DATA_BLOCK "_2010LV100P01_AD"   // DB14357
TITLE = Instance DB Adapter Block: _2010LV100P01
{ S7_Optimized_Access := 'FALSE' }
AUTHOR : METIS
NAME : APPT_DB
VERSION : 8.0
// stored: InstanceOfName IUSYS_PAC3220V1_POWERMON
"IUSYS_PAC3220V1_POWERMON"
BEGIN
   INREF := 6156;
   NET := 106;
   NODE := 22;
   RAW_InPut.SD00 := 16#0000_0001;
   RAW_InPut.SD04 := 401.1395;
   RAW_InPut.SD08 := 401.1483;
   RAW_InPut.SD12 := 400.6243;
   RAW_InPut.SD16 := 176.0122;
   RAW_InPut.SD20 := 183.3011;
   RAW_InPut.SD24 := 179.5082;
   RAW_InPut.SD28 := 49.93077;
   RAW_InPut.SD32 := 124737.3;
   RAW_InPut.SD36 := 97399.13;
   RAW_InPut.SD40 := 16734.09;
   RAW_InPut.SD44 := 0.7808338;
   RAW_InPut.SD48 := 3.005806E+08;
   RAW_InPut.SD52 := 3.817564E+08;
END_DATA_BLOCK

DATA_BLOCK "_2015PU027U01_AD"   // DB14415
{ S7_Optimized_Access := 'FALSE' }
VERSION : 0.1
// stored: InstanceOfName IUSYS_INVT_PN_MOTOR
"IUSYS_INVT_PN_MOTOR"
BEGIN
   INREF := 10040;
   OUTREF := 10040;
   FUNCTYPE := 41;
   OPTIONS := 1;
   NET := 106;
   NODE := 75;
   MCC := TRUE;
   RDY := TRUE;
   OVL := TRUE;
   LSTP := TRUE;
   REM := TRUE;
   SSW := TRUE;
   TFA := TRUE;
   DRDY := TRUE;
   STALL := TRUE;
   EARTH := TRUE;
   UBAL := TRUE;
   GFA := TRUE;
   GWA := TRUE;
   BUSF := TRUE;
   DOPR := TRUE;
   RAW_Input.SB00_0 := TRUE;
   RAW_Input.SB00_6 := TRUE;
   RAW_Input.SB01 := 16#03;
   RAW_Input.SB17_0 := TRUE;
   RAW_Input.SB17_1 := TRUE;
   RAW_Output.CB01 := 16#06;
   RAW_Output.CW08 := 16#0001;
   IHK.DelSTR_Timer_PV := 1;
   IHK.DelSTR_Timer_Mem := 1;
   IHK.DelSTP_Timer_PV := 3;
   IHK.RES_Timer_PV := 2;
   IHK.RES_Timer_Mem := 2;
   IHK.ChgOverTime_PV := 1;
   IHK.CoastTimer_PV := 1;
   IHK.DelSTP_Timer_DN := TRUE;
   IHK.ChgOverTime_DN := TRUE;
   IHK.CoastTimer_DN := TRUE;
   IHK.AUX_DelSTR_Time := 1;
   IHK.CoastSTP := TRUE;
   IHK.No_Acyc := TRUE;
   IHK.Pulse._01 := TRUE;
   IHK.Pulse._02 := TRUE;
   AC.Ons_Read_Req := TRUE;
   AC.Motor_Data_99._06 := 100.0;
   AC.Motor_Data_99._09 := 100;
   AC.Motor_Data_99._10 := 100.0;
   AC._99_Status := 16#0000_0000;
   AC_Read_99_Migra.STATUS := 16#0000_0000;
   OUT.MCC := TRUE;
   OUT.RDY := TRUE;
   OUT.OVL := TRUE;
   OUT.LSTP := TRUE;
   OUT.REM := TRUE;
   OUT.SSW := TRUE;
   OUT.TFA := TRUE;
   OUT.DRDY := TRUE;
   OUT.STALL := TRUE;
   OUT.EARTH := TRUE;
   OUT.UBAL := TRUE;
   OUT.GFA := TRUE;
   OUT.GWA := TRUE;
   OUT.BUSF := TRUE;
   OUT.DOPR := TRUE;
END_DATA_BLOCK

DATA_BLOCK "_2015PU028U01_AD"   // DB14416
{ S7_Optimized_Access := 'FALSE' }
VERSION : 0.1
// stored: InstanceOfName IUSYS_INVT_PN_MOTOR
"IUSYS_INVT_PN_MOTOR"
BEGIN
   INREF := 10072;
   OUTREF := 10072;
   FUNCTYPE := 41;
   OPTIONS := 1;
   NET := 106;
   NODE := 76;
   MCC := TRUE;
   RDY := TRUE;
   OVL := TRUE;
   REM := TRUE;
   SSW := TRUE;
   TFA := TRUE;
   DRDY := TRUE;
   STALL := TRUE;
   EARTH := TRUE;
   UBAL := TRUE;
   GFA := TRUE;
   GWA := TRUE;
   DTEST := TRUE;
   RAW_Output.CB01 := 16#06;
   RAW_Output.CW08 := 16#0001;
   IHK.DelSTR_Timer_PV := 1;
   IHK.DelSTR_Timer_Mem := 1;
   IHK.DelSTP_Timer_PV := 3;
   IHK.RES_Timer_PV := 2;
   IHK.RES_Timer_Mem := 2;
   IHK.ChgOverTime_PV := 1;
   IHK.CoastTimer_PV := 1;
   IHK.DelSTP_Timer_DN := TRUE;
   IHK.ChgOverTime_DN := TRUE;
   IHK.CoastTimer_DN := TRUE;
   IHK.AUX_DelSTR_Time := 1;
   IHK.CoastSTP := TRUE;
   IHK.No_Acyc := TRUE;
   IHK.Pulse._01 := TRUE;
   IHK.Pulse._02 := TRUE;
   AC.Ons_Read_Req := TRUE;
   AC.Motor_Data_99._06 := 100.0;
   AC.Motor_Data_99._09 := 100;
   AC.Motor_Data_99._10 := 100.0;
   AC._99_Status := 16#0000_0000;
   AC_Read_99_Migra.STATUS := 16#0000_0000;
   OUT.MCC := TRUE;
   OUT.RDY := TRUE;
   OUT.OVL := TRUE;
   OUT.REM := TRUE;
   OUT.SSW := TRUE;
   OUT.TFA := TRUE;
   OUT.DRDY := TRUE;
   OUT.STALL := TRUE;
   OUT.EARTH := TRUE;
   OUT.UBAL := TRUE;
   OUT.GFA := TRUE;
   OUT.GWA := TRUE;
   OUT.DTEST := TRUE;
END_DATA_BLOCK

DATA_BLOCK "_2015PU040U01_AD"   // DB14419
{ S7_Optimized_Access := 'FALSE' }
AUTHOR : FLSmidth
FAMILY : IUSYS
NAME : ADAPTOR
VERSION : 2.2
// stored: InstanceOfName IUSYS_ACS880_PN_MOTOR
"IUSYS_ACS880_PN_MOTOR"
BEGIN
   INREF := 10248;
   OUTREF := 10248;
   FUNCTYPE := 41;
   OPTIONS := 1;
   NET := 106;
   NODE := 16;
   CV := 100.0;
   MCC := TRUE;
   RDY := TRUE;
   OVL := TRUE;
   REM := TRUE;
   SSW := TRUE;
   TFA := TRUE;
   STALL := TRUE;
   EARTH := TRUE;
   UBAL := TRUE;
   GFA := TRUE;
   GWA := TRUE;
   BUSF := TRUE;
   DOPR := TRUE;
   RAW_Input.SB00_1 := TRUE;
   RAW_Input.SB00_4 := TRUE;
   RAW_Input.SB01_0 := TRUE;
   RAW_Input.SB01_4 := TRUE;
   RAW_Input.SB01_5 := TRUE;
   RAW_Input.SD04 := 16#0000_0000;
   RAW_Input.SD08 := 16#0000_0000;
   RAW_Input.SB16_7 := TRUE;
   RAW_Input.SW18 := 16#0B5E;
   RAW_Input.SW20 := 16#02AF;
   RAW_Output.CB00_2 := TRUE;
   RAW_Output.CB01_1 := TRUE;
   RAW_Output.CB01_2 := TRUE;
   RAW_Output.CB01_4 := TRUE;
   RAW_Output.CB01_5 := TRUE;
   RAW_Output.CB01_6 := TRUE;
   RAW_Output.CW02 := 16#4E20;
   RAW_Output.CW08 := 16#0001;
   IHK.DelSTR_Timer_PV := 1;
   IHK.DelSTR_Timer_Mem := 1;
   IHK.DelSTP_Timer_PV := 3;
   IHK.RES_Timer_PV := 2;
   IHK.RES_Timer_Mem := 2;
   IHK.ChgOverTime_PV := 1;
   IHK.CoastTimer_PV := 1;
   IHK.DelSTP_Timer_DN := TRUE;
   IHK.ChgOverTime_DN := TRUE;
   IHK.CoastTimer_DN := TRUE;
   IHK.AUX_DelSTR_Time := 1;
   IHK.CoastSTP := TRUE;
   IHK.No_Acyc := TRUE;
   IHK.Pulse._01 := TRUE;
   IHK.Pulse._02 := TRUE;
   AC.Ons_Read_Req := TRUE;
   AC._99_Status := 16#0000_0000;
   AC_Read_99_Migra.STATUS := 16#0000_0000;
   OUT.MCC := TRUE;
   OUT.RDY := TRUE;
   OUT.OVL := TRUE;
   OUT.REM := TRUE;
   OUT.SSW := TRUE;
   OUT.TFA := TRUE;
   OUT.STALL := TRUE;
   OUT.EARTH := TRUE;
   OUT.UBAL := TRUE;
   OUT.GFA := TRUE;
   OUT.GWA := TRUE;
   OUT.BUSF := TRUE;
   OUT.DOPR := TRUE;
END_DATA_BLOCK

DATA_BLOCK "_2015PU041U01_AD"   // DB14420
{ S7_Optimized_Access := 'FALSE' }
AUTHOR : FLSmidth
FAMILY : IUSYS
NAME : ADAPTOR
VERSION : 2.2
// stored: InstanceOfName IUSYS_ACS880_PN_MOTOR
"IUSYS_ACS880_PN_MOTOR"
BEGIN
   INREF := 10272;
   OUTREF := 10272;
   FUNCTYPE := 41;
   OPTIONS := 1;
   NET := 106;
   NODE := 78;
   CV := 100.0;
   MCC := TRUE;
   RDY := TRUE;
   OVL := TRUE;
   REM := TRUE;
   SSW := TRUE;
   TFA := TRUE;
   STALL := TRUE;
   EARTH := TRUE;
   UBAL := TRUE;
   GFA := TRUE;
   GWA := TRUE;
   BUSF := TRUE;
   DOPR := TRUE;
   RAW_Input.SB00_1 := TRUE;
   RAW_Input.SB00_4 := TRUE;
   RAW_Input.SB01_0 := TRUE;
   RAW_Input.SB01_4 := TRUE;
   RAW_Input.SB01_5 := TRUE;
   RAW_Input.SD04 := 16#0000_0000;
   RAW_Input.SD08 := 16#0000_0000;
   RAW_Input.SB16_7 := TRUE;
   RAW_Input.SW18 := 16#0B5E;
   RAW_Input.SW20 := 16#02AF;
   RAW_Output.CB00_2 := TRUE;
   RAW_Output.CB01_1 := TRUE;
   RAW_Output.CB01_2 := TRUE;
   RAW_Output.CB01_4 := TRUE;
   RAW_Output.CB01_5 := TRUE;
   RAW_Output.CB01_6 := TRUE;
   RAW_Output.CW02 := 16#4E20;
   RAW_Output.CW08 := 16#0001;
   IHK.DelSTR_Timer_PV := 1;
   IHK.DelSTR_Timer_Mem := 1;
   IHK.DelSTP_Timer_PV := 3;
   IHK.RES_Timer_PV := 2;
   IHK.RES_Timer_Mem := 2;
   IHK.ChgOverTime_PV := 1;
   IHK.CoastTimer_PV := 1;
   IHK.DelSTP_Timer_DN := TRUE;
   IHK.ChgOverTime_DN := TRUE;
   IHK.CoastTimer_DN := TRUE;
   IHK.AUX_DelSTR_Time := 1;
   IHK.CoastSTP := TRUE;
   IHK.No_Acyc := TRUE;
   IHK.Pulse._01 := TRUE;
   IHK.Pulse._02 := TRUE;
   AC.Ons_Read_Req := TRUE;
   AC._99_Status := 16#0000_0000;
   AC_Read_99_Migra.STATUS := 16#0000_0000;
   OUT.MCC := TRUE;
   OUT.RDY := TRUE;
   OUT.OVL := TRUE;
   OUT.REM := TRUE;
   OUT.SSW := TRUE;
   OUT.TFA := TRUE;
   OUT.STALL := TRUE;
   OUT.EARTH := TRUE;
   OUT.UBAL := TRUE;
   OUT.GFA := TRUE;
   OUT.GWA := TRUE;
   OUT.BUSF := TRUE;
   OUT.DOPR := TRUE;
END_DATA_BLOCK

DATA_BLOCK "_2015PU042U01_AD"   // DB14421
{ S7_Optimized_Access := 'FALSE' }
AUTHOR : FLSmidth
FAMILY : IUSYS
NAME : ADAPTOR
VERSION : 5.2
// stored: InstanceOfName IUSYS_3UF70_V5_MOTOR
"IUSYS_3UF70_V5_MOTOR"
BEGIN
   INREF := 7590;
   OUTREF := 7480;
   FUNCTYPE := 41;
   NET := 106;
   NODE := 64;
   MCC := TRUE;
   RDY := TRUE;
   OVL := TRUE;
   LSTP := TRUE;
   REM := TRUE;
   SSW := TRUE;
   TFA := TRUE;
   DRDY := TRUE;
   STALL := TRUE;
   EARTH := TRUE;
   UBAL := TRUE;
   GFA := TRUE;
   GWA := TRUE;
   BUSF := TRUE;
   DOPR := TRUE;
   ES := TRUE;
   Raw_InPut.SB00_1 := TRUE;
   Raw_InPut.SB00_2 := TRUE;
   Raw_InPut.SB00_3 := TRUE;
   Raw_InPut.SB01_3 := TRUE;
   Raw_OutPut.CB00_3 := TRUE;
   Raw_OutPut.CB00_7 := TRUE;
   OUT.MCC := TRUE;
   OUT.RDY := TRUE;
   OUT.OVL := TRUE;
   OUT.LSTP := TRUE;
   OUT.REM := TRUE;
   OUT.SSW := TRUE;
   OUT.TFA := TRUE;
   OUT.DRDY := TRUE;
   OUT.STALL := TRUE;
   OUT.EARTH := TRUE;
   OUT.UBAL := TRUE;
   OUT.GFA := TRUE;
   OUT.GWA := TRUE;
   OUT.BUSF := TRUE;
   OUT.DOPR := TRUE;
   OUT.ES := TRUE;
END_DATA_BLOCK

DATA_BLOCK "_MTR_SPARE_AD"   // DB14422
{ S7_Optimized_Access := 'FALSE' }
VERSION : 0.1
// stored: InstanceOfName IUSYS_ALTIVAR_PN_MOTOR
"IUSYS_ALTIVAR_PN_MOTOR"
BEGIN
END_DATA_BLOCK

DATA_BLOCK "_2015PU035U01_AD"   // DB14433
{ S7_Optimized_Access := 'FALSE' }
VERSION : 0.1
// stored: InstanceOfName IUSYS_INVT_PN_MOTOR
"IUSYS_INVT_PN_MOTOR"
BEGIN
   INREF := 10104;
   OUTREF := 10104;
   FUNCTYPE := 41;
   OPTIONS := 1;
   NET := 106;
   NODE := 75;
   CV := 20.0;
   MCC := TRUE;
   RDY := TRUE;
   OVL := TRUE;
   LSTP := TRUE;
   REM := TRUE;
   SSW := TRUE;
   TFA := TRUE;
   DRDY := TRUE;
   STALL := TRUE;
   EARTH := TRUE;
   UBAL := TRUE;
   GFA := TRUE;
   GWA := TRUE;
   BUSF := TRUE;
   DOPR := TRUE;
   RAW_Input.SB00_0 := TRUE;
   RAW_Input.SB00_6 := TRUE;
   RAW_Input.SB01 := 16#03;
   RAW_Input.SB17_0 := TRUE;
   RAW_Input.SB17_1 := TRUE;
   RAW_Output.CB01 := 16#06;
   RAW_Output.CW02 := 16#03E8;
   RAW_Output.CW08 := 16#0001;
   IHK.DelSTR_Timer_PV := 1;
   IHK.DelSTR_Timer_Mem := 1;
   IHK.DelSTP_Timer_PV := 3;
   IHK.RES_Timer_PV := 2;
   IHK.RES_Timer_Mem := 2;
   IHK.ChgOverTime_PV := 1;
   IHK.CoastTimer_PV := 1;
   IHK.DelSTP_Timer_DN := TRUE;
   IHK.ChgOverTime_DN := TRUE;
   IHK.CoastTimer_DN := TRUE;
   IHK.AUX_DelSTR_Time := 1;
   IHK.CoastSTP := TRUE;
   IHK.No_Acyc := TRUE;
   IHK.Pulse._01 := TRUE;
   IHK.Pulse._02 := TRUE;
   AC.Ons_Read_Req := TRUE;
   AC.Motor_Data_99._06 := 100.0;
   AC.Motor_Data_99._09 := 100;
   AC.Motor_Data_99._10 := 100.0;
   AC._99_Status := 16#0000_0000;
   AC_Read_99_Migra.STATUS := 16#0000_0000;
   OUT.MCC := TRUE;
   OUT.RDY := TRUE;
   OUT.OVL := TRUE;
   OUT.LSTP := TRUE;
   OUT.REM := TRUE;
   OUT.SSW := TRUE;
   OUT.TFA := TRUE;
   OUT.DRDY := TRUE;
   OUT.STALL := TRUE;
   OUT.EARTH := TRUE;
   OUT.UBAL := TRUE;
   OUT.GFA := TRUE;
   OUT.GWA := TRUE;
   OUT.BUSF := TRUE;
   OUT.DOPR := TRUE;
END_DATA_BLOCK

DATA_BLOCK "__2010CV300U01_AD"   // DB24007
{ S7_Optimized_Access := 'FALSE' }
VERSION : 0.1
// stored: InstanceOfName IUSYS_ACS880_PN_MOTOR
"IUSYS_ACS880_PN_MOTOR"
BEGIN
END_DATA_BLOCK

DATA_BLOCK "IUSYS_ALTIVAR_PN_MOTOR_DB_1"   // DB24011
{ S7_Optimized_Access := 'FALSE' }
VERSION : 0.1
// stored: InstanceOfName IUSYS_ALTIVAR_PN_MOTOR
"IUSYS_ALTIVAR_PN_MOTOR"
BEGIN
END_DATA_BLOCK

DATA_BLOCK "IUSYS_ALTIVAR_PN_MOTOR_DB"   // DB24012
{ S7_Optimized_Access := 'FALSE' }
VERSION : 0.1
// stored: InstanceOfName IUSYS_ALTIVAR_PN_MOTOR
"IUSYS_ALTIVAR_PN_MOTOR"
BEGIN
END_DATA_BLOCK

// folder: Modbus

DATA_BLOCK "MB_DATA_TEST"   // DB20
{ S7_Optimized_Access := 'FALSE' }
VERSION : 0.1
   VAR
      d12 : Word;
      d11 : Word;
      d10 : Word;
      d9 : Word;
      d8 : Word;
      d7 : Word;
      d6 : Word;
      d5 : Word;
      d4 : Word;
      d3 : Word;
      d2 : Word;
      d1 : Word;
   END_VAR
BEGIN
END_DATA_BLOCK

DATA_BLOCK "DB_DATA_MB_RD_VSD110"   // DB27
{ S7_Optimized_Access := 'FALSE' }
VERSION : 0.1
   VAR
      Frame1 : Struct
         REQ : Bool := TRUE;
         DISCONNECT : Bool := FALSE;
         CONNECT : TCON_IP_v4;
         DONE : Bool := TRUE;
         BUSY : Bool := FALSE;
         ERROR : Bool := FALSE;
         STATUS : Word := 16#0000;
         STATUS_SAVE : Word := 16#80C4;
         MB_MODE : USInt := 0;
         MB_DATA_ADDR : UDInt := 403202;
         MB_DATA_LEN : UInt := 8;
         MB_DATA_PTR : Array[0..10] of Int;
      END_STRUCT;
      Frame2 : Struct
         REQ : Bool := TRUE;
         DISCONNECT : Bool := FALSE;
         CONNECT : TCON_IP_v4;
         DONE : Bool := FALSE;
         BUSY : Bool := FALSE;
         ERROR : Bool := FALSE;
         STATUS : Word := 16#7004;
         STATUS_SAVE : Word := 16#8383;
         MB_MODE : USInt := 0;
         MB_DATA_ADDR : UDInt := 403105;
         MB_DATA_LEN : UInt := 2;
         MB_DATA_PTR : Array[0..10] of Int;
      END_STRUCT;
      Frame3 : Struct
         REQ : Bool := TRUE;
         DISCONNECT : Bool := FALSE;
         CONNECT : TCON_IP_v4;
         DONE : Bool := FALSE;
         BUSY : Bool := FALSE;
         ERROR : Bool := FALSE;
         STATUS : Word := 16#7004;
         STATUS_SAVE : Word := 16#80C6;
         MB_MODE : USInt := 0;
         MB_DATA_ADDR : UDInt := 407201;
         MB_DATA_LEN : UInt := 2;
         MB_DATA_PTR : Array[0..10] of Int;
      END_STRUCT;
      Frame4 : Struct
         REQ : Bool := TRUE;
         DISCONNECT : Bool := FALSE;
         CONNECT : TCON_IP_v4;
         DONE : Bool := FALSE;
         BUSY : Bool := FALSE;
         ERROR : Bool := FALSE;
         STATUS : Word := 16#7004;
         STATUS_SAVE : Word := 16#80C6;
         MB_MODE : USInt := 0;
         MB_DATA_ADDR : UDInt := 415323;
         MB_DATA_LEN : UInt := 2;
         MB_DATA_PTR : Array[0..10] of Int;
      END_STRUCT;
      Frame5 : Struct
         REQ : Bool := TRUE;
         DISCONNECT : Bool := FALSE;
         CONNECT : TCON_IP_v4;
         DONE : Bool := FALSE;
         BUSY : Bool := FALSE;
         ERROR : Bool := FALSE;
         STATUS : Word := 16#7000;
         STATUS_SAVE : Word := 16#8200;
         MB_MODE : USInt := 2;
         MB_DATA_ADDR : UDInt := 408502;
         MB_DATA_LEN : UInt := 2;
         MB_DATA_PTR : Array[0..10] of Int;
      END_STRUCT;
   END_VAR
BEGIN
   Frame1.CONNECT.LocalPort := 0;
   Frame1.CONNECT.RemotePort := 502;
   Frame1.CONNECT.RemoteAddress.ADDR[4] := 16#14;
   Frame1.CONNECT.RemoteAddress.ADDR[3] := 16#E7;
   Frame1.CONNECT.RemoteAddress.ADDR[2] := 16#1A;
   Frame1.CONNECT.RemoteAddress.ADDR[1] := 16#0A;
   Frame1.CONNECT.ActiveEstablished := TRUE;
   Frame1.CONNECT.ConnectionType := 16#0B;
   Frame1.CONNECT.ID := 16#0001;
   Frame1.CONNECT.InterfaceId := 64;
   Frame1.MB_DATA_PTR[0] := 3;
   Frame4.MB_DATA_PTR[10] := 0;
   Frame4.MB_DATA_PTR[9] := -32768;
   Frame4.MB_DATA_PTR[8] := 40;
   Frame4.MB_DATA_PTR[7] := 0;
   Frame4.MB_DATA_PTR[6] := 2391;
   Frame4.MB_DATA_PTR[5] := 6;
   Frame4.MB_DATA_PTR[4] := 0;
   Frame4.MB_DATA_PTR[3] := 0;
   Frame4.MB_DATA_PTR[2] := 0;
   Frame1.MB_DATA_PTR[8] := 40;
   Frame1.MB_DATA_PTR[7] := 0;
   Frame1.MB_DATA_PTR[6] := 4077;
   Frame1.MB_DATA_PTR[5] := 2;
   Frame1.MB_DATA_PTR[4] := 0;
   Frame1.MB_DATA_PTR[3] := 0;
   Frame1.MB_DATA_PTR[2] := 200;
   Frame1.MB_DATA_PTR[1] := 0;
   Frame1.MB_DATA_PTR[9] := -32768;
   Frame1.MB_DATA_PTR[10] := 0;
   Frame4.MB_DATA_PTR[1] := 0;
   Frame2.MB_DATA_PTR[10] := 0;
   Frame2.MB_DATA_PTR[9] := -32768;
   Frame2.MB_DATA_PTR[8] := 40;
   Frame2.MB_DATA_PTR[7] := 0;
   Frame2.MB_DATA_PTR[6] := 2391;
   Frame2.MB_DATA_PTR[5] := 0;
   Frame2.MB_DATA_PTR[4] := 0;
   Frame2.MB_DATA_PTR[3] := 0;
   Frame2.MB_DATA_PTR[2] := 0;
   Frame2.MB_DATA_PTR[1] := 200;
   Frame2.MB_DATA_PTR[0] := 500;
   Frame4.MB_DATA_PTR[0] := 1;
   Frame4.CONNECT.ID := 16#0004;
   Frame4.CONNECT.InterfaceId := 64;
   Frame3.MB_DATA_PTR[10] := 0;
   Frame3.MB_DATA_PTR[9] := -32768;
   Frame3.MB_DATA_PTR[8] := 40;
   Frame3.MB_DATA_PTR[7] := 0;
   Frame3.MB_DATA_PTR[6] := 2391;
   Frame3.MB_DATA_PTR[5] := 6;
   Frame3.MB_DATA_PTR[4] := 0;
   Frame3.MB_DATA_PTR[3] := 0;
   Frame3.MB_DATA_PTR[2] := 125;
   Frame3.MB_DATA_PTR[1] := 150;
   Frame3.MB_DATA_PTR[0] := 150;
   Frame4.CONNECT.LocalPort := 0;
   Frame4.CONNECT.RemotePort := 502;
   Frame4.CONNECT.RemoteAddress.ADDR[4] := 16#14;
   Frame4.CONNECT.RemoteAddress.ADDR[3] := 16#E7;
   Frame4.CONNECT.RemoteAddress.ADDR[2] := 16#1A;
   Frame4.CONNECT.RemoteAddress.ADDR[1] := 16#0A;
   Frame4.CONNECT.ActiveEstablished := TRUE;
   Frame4.CONNECT.ConnectionType := 16#0B;
   Frame2.CONNECT.LocalPort := 0;
   Frame2.CONNECT.RemotePort := 502;
   Frame2.CONNECT.RemoteAddress.ADDR[4] := 16#14;
   Frame2.CONNECT.RemoteAddress.ADDR[3] := 16#E7;
   Frame2.CONNECT.RemoteAddress.ADDR[2] := 16#1A;
   Frame2.CONNECT.RemoteAddress.ADDR[1] := 16#0A;
   Frame2.CONNECT.ActiveEstablished := TRUE;
   Frame2.CONNECT.ConnectionType := 16#0B;
   Frame2.CONNECT.ID := 16#0002;
   Frame2.CONNECT.InterfaceId := 64;
   Frame3.CONNECT.LocalPort := 0;
   Frame3.CONNECT.RemotePort := 502;
   Frame3.CONNECT.RemoteAddress.ADDR[4] := 16#14;
   Frame3.CONNECT.RemoteAddress.ADDR[3] := 16#E7;
   Frame3.CONNECT.RemoteAddress.ADDR[2] := 16#1A;
   Frame3.CONNECT.RemoteAddress.ADDR[1] := 16#0A;
   Frame3.CONNECT.ActiveEstablished := TRUE;
   Frame3.CONNECT.ConnectionType := 16#0B;
   Frame3.CONNECT.ID := 16#0003;
   Frame3.CONNECT.InterfaceId := 64;
   Frame5.CONNECT.InterfaceId := 64;
   Frame5.CONNECT.ID := 16#0005;
   Frame5.CONNECT.ConnectionType := 16#0B;
   Frame5.CONNECT.ActiveEstablished := TRUE;
   Frame5.CONNECT.RemoteAddress.ADDR[1] := 16#0A;
   Frame5.CONNECT.RemoteAddress.ADDR[2] := 16#1A;
   Frame5.CONNECT.RemoteAddress.ADDR[3] := 16#E7;
   Frame5.CONNECT.RemoteAddress.ADDR[4] := 16#14;
   Frame5.CONNECT.RemotePort := 502;
   Frame5.CONNECT.LocalPort := 0;
   Frame5.MB_DATA_PTR[0] := 0;
   Frame5.MB_DATA_PTR[1] := 125;
   Frame5.MB_DATA_PTR[2] := 125;
   Frame5.MB_DATA_PTR[3] := 0;
   Frame5.MB_DATA_PTR[4] := 0;
   Frame5.MB_DATA_PTR[5] := 6;
   Frame5.MB_DATA_PTR[6] := 2391;
   Frame5.MB_DATA_PTR[7] := 0;
   Frame5.MB_DATA_PTR[8] := 40;
   Frame5.MB_DATA_PTR[9] := -32768;
   Frame5.MB_DATA_PTR[10] := 0;
END_DATA_BLOCK

DATA_BLOCK "DB_DATA_MB_RD_VSD130_t"   // DB28
{ S7_Optimized_Access := 'FALSE' }
VERSION : 0.1
   VAR
      Frame1 : Struct
         REQ : Bool := TRUE;
         DISCONNECT : Bool := FALSE;
         CONNECT : TCON_IP_v4;
         DONE : Bool := FALSE;
         BUSY : Bool := FALSE;
         ERROR : Bool := FALSE;
         STATUS : Word := 16#7000;
         STATUS_SAVE : Word := 16#80C4;
         MB_MODE : USInt := 0;
         MB_DATA_ADDR : UDInt := 403202;
         MB_DATA_LEN : UInt := 8;
         MB_DATA_PTR : Array[0..10] of Int;
      END_STRUCT;
      Frame2 : Struct
         REQ : Bool := TRUE;
         DISCONNECT : Bool := FALSE;
         CONNECT : TCON_IP_v4;
         DONE : Bool := FALSE;
         BUSY : Bool := FALSE;
         ERROR : Bool := FALSE;
         STATUS : Word := 16#7000;
         STATUS_SAVE : Word := 16#80C6;
         MB_MODE : USInt := 0;
         MB_DATA_ADDR : UDInt := 403105;
         MB_DATA_LEN : UInt := 2;
         MB_DATA_PTR : Array[0..10] of Int;
      END_STRUCT;
      Frame3 : Struct
         REQ : Bool := FALSE;
         DISCONNECT : Bool := FALSE;
         CONNECT : TCON_IP_v4;
         DONE : Bool := FALSE;
         BUSY : Bool := FALSE;
         ERROR : Bool := FALSE;
         STATUS : Word := 16#7000;
         STATUS_SAVE : Word := 16#80C6;
         MB_MODE : USInt := 0;
         MB_DATA_ADDR : UDInt := 407201;
         MB_DATA_LEN : UInt := 2;
         MB_DATA_PTR : Array[0..10] of Int;
      END_STRUCT;
      Frame4 : Struct
         REQ : Bool := TRUE;
         DISCONNECT : Bool := FALSE;
         CONNECT : TCON_IP_v4;
         DONE : Bool := FALSE;
         BUSY : Bool := FALSE;
         ERROR : Bool := FALSE;
         STATUS : Word := 16#7000;
         STATUS_SAVE : Word := 16#80C6;
         MB_MODE : USInt := 0;
         MB_DATA_ADDR : UDInt := 415323;
         MB_DATA_LEN : UInt := 2;
         MB_DATA_PTR : Array[0..10] of Int;
      END_STRUCT;
      Frame5 : Struct
         REQ : Bool := TRUE;
         DISCONNECT : Bool := FALSE;
         CONNECT : TCON_IP_v4;
         DONE : Bool := FALSE;
         BUSY : Bool := FALSE;
         ERROR : Bool := FALSE;
         STATUS : Word := 16#7002;
         STATUS_SAVE : Word := 16#80C6;
         MB_MODE : USInt := 2;
         MB_DATA_ADDR : UDInt := 408502;
         MB_DATA_LEN : UInt := 2;
         MB_DATA_PTR : Array[0..10] of Int;
      END_STRUCT;
   END_VAR
BEGIN
   Frame1.CONNECT.LocalPort := 0;
   Frame1.CONNECT.RemotePort := 502;
   Frame1.CONNECT.RemoteAddress.ADDR[4] := 16#16;
   Frame1.CONNECT.RemoteAddress.ADDR[3] := 16#E7;
   Frame1.CONNECT.RemoteAddress.ADDR[2] := 16#1A;
   Frame1.CONNECT.RemoteAddress.ADDR[1] := 16#0A;
   Frame1.CONNECT.ActiveEstablished := TRUE;
   Frame1.CONNECT.ConnectionType := 16#0B;
   Frame1.CONNECT.ID := 16#0006;
   Frame1.CONNECT.InterfaceId := 64;
   Frame1.MB_DATA_PTR[0] := 545;
   Frame4.MB_DATA_PTR[10] := 0;
   Frame4.MB_DATA_PTR[9] := -32768;
   Frame4.MB_DATA_PTR[8] := 40;
   Frame4.MB_DATA_PTR[7] := 0;
   Frame4.MB_DATA_PTR[6] := 2391;
   Frame4.MB_DATA_PTR[5] := 6;
   Frame4.MB_DATA_PTR[4] := 0;
   Frame4.MB_DATA_PTR[3] := 0;
   Frame4.MB_DATA_PTR[2] := 0;
   Frame1.MB_DATA_PTR[8] := 0;
   Frame1.MB_DATA_PTR[7] := 0;
   Frame1.MB_DATA_PTR[6] := 0;
   Frame1.MB_DATA_PTR[5] := 2;
   Frame1.MB_DATA_PTR[4] := 0;
   Frame1.MB_DATA_PTR[3] := 0;
   Frame1.MB_DATA_PTR[2] := 500;
   Frame1.MB_DATA_PTR[1] := 0;
   Frame1.MB_DATA_PTR[9] := 0;
   Frame1.MB_DATA_PTR[10] := 0;
   Frame4.MB_DATA_PTR[1] := 3;
   Frame2.MB_DATA_PTR[10] := 0;
   Frame2.MB_DATA_PTR[9] := -32768;
   Frame2.MB_DATA_PTR[8] := 40;
   Frame2.MB_DATA_PTR[7] := 0;
   Frame2.MB_DATA_PTR[6] := 2391;
   Frame2.MB_DATA_PTR[5] := 0;
   Frame2.MB_DATA_PTR[4] := 0;
   Frame2.MB_DATA_PTR[3] := 0;
   Frame2.MB_DATA_PTR[2] := 0;
   Frame2.MB_DATA_PTR[1] := 0;
   Frame2.MB_DATA_PTR[0] := 500;
   Frame4.MB_DATA_PTR[0] := 0;
   Frame4.CONNECT.ID := 16#0009;
   Frame4.CONNECT.InterfaceId := 64;
   Frame3.MB_DATA_PTR[10] := 0;
   Frame3.MB_DATA_PTR[9] := -32768;
   Frame3.MB_DATA_PTR[8] := 40;
   Frame3.MB_DATA_PTR[7] := 0;
   Frame3.MB_DATA_PTR[6] := 0;
   Frame3.MB_DATA_PTR[5] := 6;
   Frame3.MB_DATA_PTR[4] := 0;
   Frame3.MB_DATA_PTR[3] := 0;
   Frame3.MB_DATA_PTR[2] := 0;
   Frame3.MB_DATA_PTR[1] := 150;
   Frame3.MB_DATA_PTR[0] := 0;
   Frame4.CONNECT.LocalPort := 0;
   Frame4.CONNECT.RemotePort := 502;
   Frame4.CONNECT.RemoteAddress.ADDR[4] := 16#16;
   Frame4.CONNECT.RemoteAddress.ADDR[3] := 16#E7;
   Frame4.CONNECT.RemoteAddress.ADDR[2] := 16#1A;
   Frame4.CONNECT.RemoteAddress.ADDR[1] := 16#0A;
   Frame4.CONNECT.ActiveEstablished := TRUE;
   Frame4.CONNECT.ConnectionType := 16#0B;
   Frame2.CONNECT.LocalPort := 0;
   Frame2.CONNECT.RemotePort := 502;
   Frame2.CONNECT.RemoteAddress.ADDR[4] := 16#16;
   Frame2.CONNECT.RemoteAddress.ADDR[3] := 16#E7;
   Frame2.CONNECT.RemoteAddress.ADDR[2] := 16#1A;
   Frame2.CONNECT.RemoteAddress.ADDR[1] := 16#0A;
   Frame2.CONNECT.ActiveEstablished := TRUE;
   Frame2.CONNECT.ConnectionType := 16#0B;
   Frame2.CONNECT.ID := 16#0007;
   Frame2.CONNECT.InterfaceId := 64;
   Frame3.CONNECT.LocalPort := 0;
   Frame3.CONNECT.RemotePort := 502;
   Frame3.CONNECT.RemoteAddress.ADDR[4] := 16#16;
   Frame3.CONNECT.RemoteAddress.ADDR[3] := 16#E7;
   Frame3.CONNECT.RemoteAddress.ADDR[2] := 16#1A;
   Frame3.CONNECT.RemoteAddress.ADDR[1] := 16#0A;
   Frame3.CONNECT.ActiveEstablished := TRUE;
   Frame3.CONNECT.ConnectionType := 16#0B;
   Frame3.CONNECT.ID := 16#0008;
   Frame3.CONNECT.InterfaceId := 64;
   Frame5.CONNECT.InterfaceId := 64;
   Frame5.CONNECT.ID := 16#000A;
   Frame5.CONNECT.ConnectionType := 16#0B;
   Frame5.CONNECT.ActiveEstablished := TRUE;
   Frame5.CONNECT.RemoteAddress.ADDR[1] := 16#0A;
   Frame5.CONNECT.RemoteAddress.ADDR[2] := 16#1A;
   Frame5.CONNECT.RemoteAddress.ADDR[3] := 16#E7;
   Frame5.CONNECT.RemoteAddress.ADDR[4] := 16#16;
   Frame5.CONNECT.RemotePort := 502;
   Frame5.CONNECT.LocalPort := 0;
   Frame5.MB_DATA_PTR[0] := 0;
   Frame5.MB_DATA_PTR[1] := 500;
   Frame5.MB_DATA_PTR[2] := 0;
   Frame5.MB_DATA_PTR[3] := 0;
   Frame5.MB_DATA_PTR[4] := 0;
   Frame5.MB_DATA_PTR[5] := 6;
   Frame5.MB_DATA_PTR[6] := 2391;
   Frame5.MB_DATA_PTR[7] := 0;
   Frame5.MB_DATA_PTR[8] := 40;
   Frame5.MB_DATA_PTR[9] := -32768;
   Frame5.MB_DATA_PTR[10] := 0;
END_DATA_BLOCK

DATA_BLOCK "VSD110"   // DB29
{ S7_Optimized_Access := 'TRUE' }
VERSION : 0.1
// stored: InstanceOfName Mgt_VSD_Com
"Mgt_VSD_Com"
BEGIN
   "Counter".CU := TRUE;
   "Counter".R := TRUE;
   "Counter".QD := TRUE;
   "Counter".PV := 1;
   Time_Value2 := 50;
   Time_Value3 := 50;
   Time_Value4 := 50;
   Time_Value5 := 50;
   Time_Value6 := 50;
   Time_Value7 := 50;
   Time_Value8 := 50;
   Time_Value9 := 50;
END_DATA_BLOCK

DATA_BLOCK "VSD130_t"   // DB30
{ S7_Optimized_Access := 'TRUE' }
VERSION : 0.1
// stored: InstanceOfName Mgt_VSD_Com
"Mgt_VSD_Com"
BEGIN
   "Counter".CU := TRUE;
   "Counter".R := TRUE;
   "Counter".QD := TRUE;
   "Counter".PV := 1;
   Time_Value2 := 50;
   Time_Value3 := 50;
   Time_Value4 := 50;
   Time_Value5 := 50;
   Time_Value6 := 50;
   Time_Value7 := 50;
   Time_Value8 := 50;
   Time_Value9 := 50;
   RD_3201_3208.MB_DATA_ADDR := 400001;
   RD_3201_3208.MB_DATA_LEN := 4;
   RD_3201_3208.STATUS := 16#7004;
   RD_3104_3105.MB_DATA_ADDR := 400004;
   RD_3104_3105.MB_DATA_LEN := 2;
   RD_3104_3105.STATUS := 16#7004;
   RD_7200_7201.MB_DATA_ADDR := 400005;
   RD_7200_7201.MB_DATA_LEN := 2;
   RD_7200_7201.STATUS := 16#7004;
   RD_15323.REQ := TRUE;
   RD_15323.MB_DATA_ADDR := 400007;
   RD_15323.MB_DATA_LEN := 2;
   RD_15323.BUSY := TRUE;
   RD_15323.STATUS := 16#7006;
   WR_8501_8502.DISCONNECT := TRUE;
   WR_8501_8502.MB_MODE := 2;
   WR_8501_8502.MB_DATA_ADDR := 40008;
   WR_8501_8502.MB_DATA_LEN := 2;
   WR_8501_8502.STATUS := 16#7000;
END_DATA_BLOCK

DATA_BLOCK "DB_DATA_MB_RD_VSD130"   // DB31
{ S7_Optimized_Access := 'FALSE' }
VERSION : 0.1
   VAR
      Frame1 : Struct
         REQ : Bool := TRUE;
         DISCONNECT : Bool := FALSE;
         CONNECT : TCON_IP_v4;
         DONE : Bool := FALSE;
         BUSY : Bool := FALSE;
         ERROR : Bool := FALSE;
         STATUS : Word := 16#7004;
         STATUS_SAVE : Word := 16#8383;
         MB_MODE : USInt := 0;
         MB_DATA_ADDR : UDInt := 403202;
         MB_DATA_LEN : UInt := 8;
         MB_DATA_PTR : Array[0..10] of Int;
      END_STRUCT;
      Frame2 : Struct
         REQ : Bool := TRUE;
         DISCONNECT : Bool := FALSE;
         CONNECT : TCON_IP_v4;
         DONE : Bool := FALSE;
         BUSY : Bool := FALSE;
         ERROR : Bool := FALSE;
         STATUS : Word := 16#7004;
         STATUS_SAVE : Word := 16#8383;
         MB_MODE : USInt := 0;
         MB_DATA_ADDR : UDInt := 403105;
         MB_DATA_LEN : UInt := 2;
         MB_DATA_PTR : Array[0..10] of Int;
      END_STRUCT;
      Frame3 : Struct
         REQ : Bool := TRUE;
         DISCONNECT : Bool := FALSE;
         CONNECT : TCON_IP_v4;
         DONE : Bool := TRUE;
         BUSY : Bool := FALSE;
         ERROR : Bool := FALSE;
         STATUS : Word := 16#0000;
         STATUS_SAVE : Word := 16#8383;
         MB_MODE : USInt := 0;
         MB_DATA_ADDR : UDInt := 407201;
         MB_DATA_LEN : UInt := 2;
         MB_DATA_PTR : Array[0..10] of Int;
      END_STRUCT;
      Frame4 : Struct
         REQ : Bool := TRUE;
         DISCONNECT : Bool := FALSE;
         CONNECT : TCON_IP_v4;
         DONE : Bool := FALSE;
         BUSY : Bool := FALSE;
         ERROR : Bool := FALSE;
         STATUS : Word := 16#7004;
         STATUS_SAVE : Word := 16#8383;
         MB_MODE : USInt := 0;
         MB_DATA_ADDR : UDInt := 415323;
         MB_DATA_LEN : UInt := 2;
         MB_DATA_PTR : Array[0..10] of Int;
      END_STRUCT;
      Frame5 : Struct
         REQ : Bool := TRUE;
         DISCONNECT : Bool := FALSE;
         CONNECT : TCON_IP_v4;
         DONE : Bool := FALSE;
         BUSY : Bool := FALSE;
         ERROR : Bool := FALSE;
         STATUS : Word := 16#7000;
         STATUS_SAVE : Word := 16#80C4;
         MB_MODE : USInt := 2;
         MB_DATA_ADDR : UDInt := 408502;
         MB_DATA_LEN : UInt := 2;
         MB_DATA_PTR : Array[0..10] of Int;
      END_STRUCT;
   END_VAR
BEGIN
   Frame1.CONNECT.LocalPort := 0;
   Frame1.CONNECT.RemotePort := 502;
   Frame1.CONNECT.RemoteAddress.ADDR[4] := 16#16;
   Frame1.CONNECT.RemoteAddress.ADDR[3] := 16#E7;
   Frame1.CONNECT.RemoteAddress.ADDR[2] := 16#1A;
   Frame1.CONNECT.RemoteAddress.ADDR[1] := 16#0A;
   Frame1.CONNECT.ActiveEstablished := TRUE;
   Frame1.CONNECT.ConnectionType := 16#0B;
   Frame1.CONNECT.ID := 16#0006;
   Frame1.CONNECT.InterfaceId := 64;
   Frame1.MB_DATA_PTR[0] := 545;
   Frame4.MB_DATA_PTR[10] := 0;
   Frame4.MB_DATA_PTR[9] := -32768;
   Frame4.MB_DATA_PTR[8] := 40;
   Frame4.MB_DATA_PTR[7] := 0;
   Frame4.MB_DATA_PTR[6] := 2391;
   Frame4.MB_DATA_PTR[5] := 6;
   Frame4.MB_DATA_PTR[4] := 0;
   Frame4.MB_DATA_PTR[3] := 0;
   Frame4.MB_DATA_PTR[2] := 0;
   Frame1.MB_DATA_PTR[8] := 40;
   Frame1.MB_DATA_PTR[7] := 0;
   Frame1.MB_DATA_PTR[6] := 0;
   Frame1.MB_DATA_PTR[5] := 2;
   Frame1.MB_DATA_PTR[4] := 0;
   Frame1.MB_DATA_PTR[3] := 0;
   Frame1.MB_DATA_PTR[2] := 500;
   Frame1.MB_DATA_PTR[1] := 0;
   Frame1.MB_DATA_PTR[9] := -32768;
   Frame1.MB_DATA_PTR[10] := 0;
   Frame4.MB_DATA_PTR[1] := 3;
   Frame2.MB_DATA_PTR[10] := 0;
   Frame2.MB_DATA_PTR[9] := -32768;
   Frame2.MB_DATA_PTR[8] := 40;
   Frame2.MB_DATA_PTR[7] := 0;
   Frame2.MB_DATA_PTR[6] := 2391;
   Frame2.MB_DATA_PTR[5] := 0;
   Frame2.MB_DATA_PTR[4] := 0;
   Frame2.MB_DATA_PTR[3] := 0;
   Frame2.MB_DATA_PTR[2] := 0;
   Frame2.MB_DATA_PTR[1] := 0;
   Frame2.MB_DATA_PTR[0] := 500;
   Frame4.MB_DATA_PTR[0] := 0;
   Frame4.CONNECT.ID := 16#0009;
   Frame4.CONNECT.InterfaceId := 64;
   Frame3.MB_DATA_PTR[10] := 0;
   Frame3.MB_DATA_PTR[9] := -32768;
   Frame3.MB_DATA_PTR[8] := 40;
   Frame3.MB_DATA_PTR[7] := 0;
   Frame3.MB_DATA_PTR[6] := 2391;
   Frame3.MB_DATA_PTR[5] := 6;
   Frame3.MB_DATA_PTR[4] := 0;
   Frame3.MB_DATA_PTR[3] := 0;
   Frame3.MB_DATA_PTR[2] := 125;
   Frame3.MB_DATA_PTR[1] := 150;
   Frame3.MB_DATA_PTR[0] := 0;
   Frame4.CONNECT.LocalPort := 0;
   Frame4.CONNECT.RemotePort := 502;
   Frame4.CONNECT.RemoteAddress.ADDR[4] := 16#16;
   Frame4.CONNECT.RemoteAddress.ADDR[3] := 16#E7;
   Frame4.CONNECT.RemoteAddress.ADDR[2] := 16#1A;
   Frame4.CONNECT.RemoteAddress.ADDR[1] := 16#0A;
   Frame4.CONNECT.ActiveEstablished := TRUE;
   Frame4.CONNECT.ConnectionType := 16#0B;
   Frame2.CONNECT.LocalPort := 0;
   Frame2.CONNECT.RemotePort := 502;
   Frame2.CONNECT.RemoteAddress.ADDR[4] := 16#16;
   Frame2.CONNECT.RemoteAddress.ADDR[3] := 16#E7;
   Frame2.CONNECT.RemoteAddress.ADDR[2] := 16#1A;
   Frame2.CONNECT.RemoteAddress.ADDR[1] := 16#0A;
   Frame2.CONNECT.ActiveEstablished := TRUE;
   Frame2.CONNECT.ConnectionType := 16#0B;
   Frame2.CONNECT.ID := 16#0007;
   Frame2.CONNECT.InterfaceId := 64;
   Frame3.CONNECT.LocalPort := 0;
   Frame3.CONNECT.RemotePort := 502;
   Frame3.CONNECT.RemoteAddress.ADDR[4] := 16#16;
   Frame3.CONNECT.RemoteAddress.ADDR[3] := 16#E7;
   Frame3.CONNECT.RemoteAddress.ADDR[2] := 16#1A;
   Frame3.CONNECT.RemoteAddress.ADDR[1] := 16#0A;
   Frame3.CONNECT.ActiveEstablished := TRUE;
   Frame3.CONNECT.ConnectionType := 16#0B;
   Frame3.CONNECT.ID := 16#0008;
   Frame3.CONNECT.InterfaceId := 64;
   Frame5.CONNECT.InterfaceId := 64;
   Frame5.CONNECT.ID := 16#000A;
   Frame5.CONNECT.ConnectionType := 16#0B;
   Frame5.CONNECT.ActiveEstablished := TRUE;
   Frame5.CONNECT.RemoteAddress.ADDR[1] := 16#0A;
   Frame5.CONNECT.RemoteAddress.ADDR[2] := 16#1A;
   Frame5.CONNECT.RemoteAddress.ADDR[3] := 16#E7;
   Frame5.CONNECT.RemoteAddress.ADDR[4] := 16#16;
   Frame5.CONNECT.RemotePort := 502;
   Frame5.CONNECT.LocalPort := 0;
   Frame5.MB_DATA_PTR[0] := 0;
   Frame5.MB_DATA_PTR[1] := 500;
   Frame5.MB_DATA_PTR[2] := 125;
   Frame5.MB_DATA_PTR[3] := 0;
   Frame5.MB_DATA_PTR[4] := 0;
   Frame5.MB_DATA_PTR[5] := 6;
   Frame5.MB_DATA_PTR[6] := 2391;
   Frame5.MB_DATA_PTR[7] := 0;
   Frame5.MB_DATA_PTR[8] := 40;
   Frame5.MB_DATA_PTR[9] := -32768;
   Frame5.MB_DATA_PTR[10] := 0;
END_DATA_BLOCK

DATA_BLOCK "VSD130_DB"   // DB32
{ S7_Optimized_Access := 'TRUE' }
VERSION : 0.1
// stored: InstanceOfName Mgt_VSD_Com
"Mgt_VSD_Com"
BEGIN
END_DATA_BLOCK

// folder: System blocks/Program resources

DATA_BLOCK "Speed_BC180_1"   // DB19
{ S7_Optimized_Access := 'TRUE' }
AUTHOR : Simatic
FAMILY : IEC
NAME : IEC_TMR
VERSION : 1.0
// stored: InstanceOfName IEC_TIMER
"IEC_TIMER"
BEGIN
END_DATA_BLOCK

DATA_BLOCK "Speed_BC180_2"   // DB21
{ S7_Optimized_Access := 'TRUE' }
AUTHOR : Simatic
FAMILY : IEC
NAME : IEC_TMR
VERSION : 1.0
// stored: InstanceOfName IEC_TIMER
"IEC_TIMER"
BEGIN
END_DATA_BLOCK

DATA_BLOCK "Speed_BC120_1"   // DB22
{ S7_Optimized_Access := 'TRUE' }
AUTHOR : Simatic
FAMILY : IEC
NAME : IEC_TMR
VERSION : 1.0
// stored: InstanceOfName IEC_TIMER
"IEC_TIMER"
BEGIN
END_DATA_BLOCK

DATA_BLOCK "Speed_BC120_2"   // DB23
{ S7_Optimized_Access := 'TRUE' }
AUTHOR : Simatic
FAMILY : IEC
NAME : IEC_TMR
VERSION : 1.0
// stored: InstanceOfName IEC_TIMER
"IEC_TIMER"
BEGIN
END_DATA_BLOCK

DATA_BLOCK "_2010SJ950M01_T1"   // DB24
{ S7_Optimized_Access := 'TRUE' }
AUTHOR : Simatic
FAMILY : IEC
NAME : IEC_TMR
VERSION : 1.0
// stored: InstanceOfName IEC_TIMER
"IEC_TIMER"
BEGIN
END_DATA_BLOCK

DATA_BLOCK "IEC_Timer_0_DB"   // DB50
{ S7_Optimized_Access := 'TRUE' }
AUTHOR : Simatic
FAMILY : IEC
NAME : IEC_TMR
VERSION : 1.0
// stored: InstanceOfName IEC_TIMER
"IEC_TIMER"
BEGIN
   ST := T#20D_8H_56M_38S_289MS;
   PT := T#2S;
END_DATA_BLOCK

// folder: (top level)

FUNCTION_BLOCK "LMNGEN_C"   // FB33, LAD
TITLE = PID : Output continuous PID controller
{ S7_Optimized_Access := 'FALSE' }
AUTHOR : MODIFIED
FAMILY : MODCONT
NAME : LMNGEN_C
VERSION : 1.0
   VAR_INPUT
      MAN : Real;   // manual value
      LMN_HLM : Real := 100.0;   // manipulated value high limit
      LMN_LLM : Real;   // manipulated value low limit
      LMN_URLM : Real := 10.0;   // manipulated value up rate limit
      LMN_DRLM : Real := 10.0;   // manipulated down rate limit
      DF_OUTV : Real;   // default output variable
      MAN_ON : Bool := TRUE;   // manual value on
      MANGN_ON : Bool;   // manual value generating on
      MANUP : Bool;   // manual value up
      MANDN : Bool;   // manual value down
      LMNRC_ON : Bool;   // manipulated value rate of change on
      DFOUT_ON : Bool;   // default output variable on
      COM_RST : Bool;   // complete restart
      CYCLE : Time := T#1S;   // sample time
      PID_LMNG : Struct
         PID_OUTV : Real;   // PID output variable
         PID_SCTR : Real;   // PID output variable for step controller
      END_STRUCT;
   END_VAR
   VAR_OUTPUT
      LMN : Real;   // manipulated value
      QLMN_HLM : Bool;   // high limit of manipulated value reached
      QLMN_LLM : Bool;   // low limit of manipulated value reached
      LMNG_PID : Struct
         LMN : Real;   // manipulated value
         LMN_HLM : Real;   // manipulated value high limit
         LMN_LLM : Real;   // manipulated value low limit
         R_MTR_TM : Real;   // motor manipulated value
         ARWHL_ON : Bool;   // anti reset wind-up in high limit on
         ARWLL_ON : Bool;   // anti reset wind-up in low limit on
         MAN_ON : Bool;   // manual mode on
         LMNGS_ON : Bool;   // PID-algorithm for step controller on
         LMNR_ON : Bool;   // repeated manipulated value on
      END_STRUCT;
   END_VAR
   VAR
      MP1 : Real;   // MP1: manipulated value
      LMN_OP : Real;   // manipulated value operation
      LMNOP_ON : Bool;   // manipulated value operation on
      stUpMan : Time;
      stDownMan : Time;
   END_VAR
   VAR_TEMP
      Hvar : Real;   // Hilfsvariable
      rCycle : Real;   // Abtastzeit in real
      Diff : Real;   // Änderungswert bei der Handwertbedienung
      RocHlm : Real;   // Obere Begrenzung im Hochlaufgeber
      RocLlm : Real;   // Untere Begrenzung im Hochlaufgeber
      Pid_Outv : Real;   // PID output variable
      dLmn : Real;   // Stellwert
      bLmnopOn : Bool;   // manipulated value operation on
      bCasOn : Bool;   // cascade mode on
      bArwhlOn : Bool;   // Anti Reset Wind-up high limit Bit für Struktur PID_LMNG
      bArwllOn : Bool;   // Anti Reset Wind-up low limit Bit für Struktur PID_LMNG
   END_VAR
BEGIN
END_FUNCTION_BLOCK

FUNCTION_BLOCK "PID"   // FB39, LAD
TITLE = PID: Output PID-algorithm
{ S7_Optimized_Access := 'FALSE' }
AUTHOR : MODIFIED
FAMILY : MODCONT
NAME : PID
VERSION : 1.1
   VAR_INPUT
      ER : Real;   // error-signal
      PV : Real;   // process variable
      GAIN : Real := 1.0;   // proportional gain
      TI : Time := T#20S;   // reset time
      I_ITLVAL : Real;   // initialization value of the integral action
      TD : Time := T#10S;   // derivative time
      TM_LAG : Time := T#2S;   // time lag of the derivative action
      DISV : Real;   // disturbance variable
      P_SEL : Bool := TRUE;   // proportional action selected
      PFDB_SEL : Bool;   // proportional action in feedback path selected
      DFDB_SEL : Bool;   // derivative action in feedback path on
      I_SEL : Bool := TRUE;   // integral action selected
      INT_HOLD : Bool;   // integral action hold
      I_ITL_ON : Bool;   // initialization of the integral action on
      D_SEL : Bool;   // derivative action selected
      DISV_SEL : Bool := TRUE;   // disturbance variable on
      COM_RST : Bool;   // complete restart
      CYCLE : Time := T#1S;   // sample time
      LMNG_PID : Struct
         LMN : Real;   // manipulated value
         LMN_HLM : Real;   // manipulated value high limit
         LMN_LLM : Real;   // manipulated value low limit
         R_MTR_TM : Real;   // motor manipulated value
         ARWHL_ON : Bool;   // anti reset wind-up in high limit on
         ARWLL_ON : Bool;   // anti reset wind-up in low limit on
         MAN_ON : Bool;   // manual mode on
         LMNGS_ON : Bool;   // PID-algorithm for step controller on
         LMNR_ON : Bool;   // repeated manipulated value on
      END_STRUCT;
   END_VAR
   VAR_OUTPUT
      LMN_P : Real;   // proportionality component
      LMN_I : Real;   // integral component
      LMN_D : Real;   // derivative component
      PID_LMNG : Struct
         PID_OUTV : Real;   // PID output variable
         PID_SCTR : Real;   // PID output variable for step controller
      END_STRUCT;
   END_VAR
   VAR
      sInvAlt : Real;
      sIanteilAlt : Real;
      sRestInt : Real;
      sRestDif : Real;
      sRueck : Real;
      sbILimOn : Bool := TRUE;
   END_VAR
   VAR_TEMP
      Hvar : Real;   // Hilfsvariable
      ErKp : Real;   // Variable ER*GAIN
      rTi : Real;   // Integrationszeit in real
      rTd : Real;   // Differentiationszeit in real
      rTmLag : Real;   // Verzögerungszeit in real
      rCycle : Real;   // Abtastzeit in real
      Panteil : Real;   // P-Anteil
      Ianteil : Real;   // I-Anteil
      Diff : Real;   // Änderungswert
      Danteil : Real;   // D-Anteil
      Verstaerk : Real;   // Verstärkung
      RueckDiff : Real;   // Differenz des Rückkopplungswertes
      RueckAlt : Real;   // Alter Rückkopplungswert
      dDisv : Real;   // disturbance variable
      dLmn : Real;   // Stellwert
      PidOutv : Real;   // PID-Ausgangswert
      PidSctr : Real;   // PID-Ausgangswert für Schrittregler
      rLmnHlm : Real;   // Obere Begrenzung
      rLmnLlm : Real;   // Untere Begrenzung
      rMtrTm : Real;   // Motorstellzeit
      bArwhlOn : Bool;   // anti reset wind-up in high limit on
      bArwllOn : Bool;   // anti reset wind-up in low limit on
      bManOn : Bool;   // manual mode on
      bLmngsOn : Bool;   // PID-algorithm for step controller
      bLmnrOn : Bool;   // step controller with repeated manipulated value
   END_VAR
BEGIN
END_FUNCTION_BLOCK

FUNCTION_BLOCK "Eqip_Maintenance"   // FB106, FBD
TITLE = Equipment Maintenance Hour Meter (5 sec)
{ S7_Optimized_Access := 'FALSE' }
VERSION : 0.1
   VAR_INPUT
      IN : Bool;   // Equipment (Motor) Status
      Reset_1 : Bool;   // Maintenance Done
      Reset_2 : Bool;   // Maintenance Done
      Reset_3 : Bool;   // Maintenance Done
      Reset_4 : Bool;   // Maintenance Done
   END_VAR
   VAR_OUTPUT
      Cnt_Hours_1 : DInt;   // Counter-1 of Hours
      Cnt_Hours_2 : DInt;   // Counter-2 of Hours
      Cnt_Hours_3 : DInt;   // Counter-3 of Hours
      Cnt_Hours_4 : DInt;   // Counter-4 of Hours
   END_VAR
   VAR
      Accum_1 : DInt;   // Accum_1 (sec)
      Accum_2 : DInt;   // Accum_2 (sec)
      Accum_3 : DInt;   // Accum_3 (sec)
      Accum_4 : DInt;   // Accum_4 (sec)
   END_VAR
   VAR_TEMP
      tmp_bool : Bool;
   END_VAR
BEGIN

REGION Network 1: Reset Seconds ACCUM_1
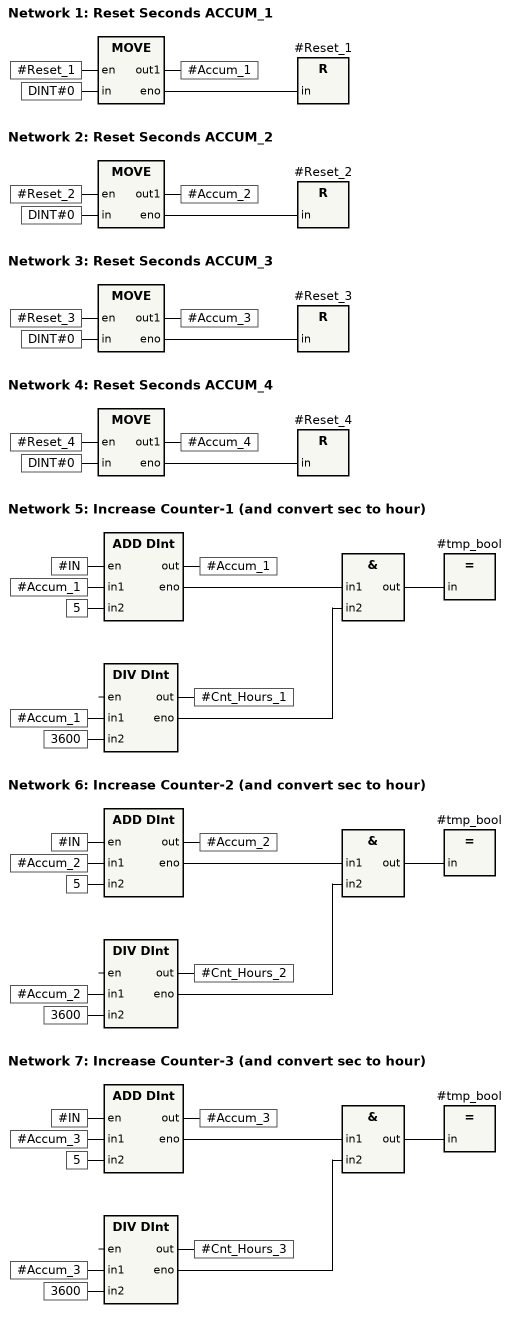
   IF #Reset_1 THEN
       #Accum_1 := DINT#0;
       #Reset_1 := FALSE;
   END_IF;
END_REGION

REGION Network 2: Reset Seconds ACCUM_2
   IF #Reset_2 THEN
       #Accum_2 := DINT#0;
       #Reset_2 := FALSE;
   END_IF;
END_REGION

REGION Network 3: Reset Seconds ACCUM_3
   IF #Reset_3 THEN
       #Accum_3 := DINT#0;
       #Reset_3 := FALSE;
   END_IF;
END_REGION

REGION Network 4: Reset Seconds ACCUM_4
   IF #Reset_4 THEN
       #Accum_4 := DINT#0;
       #Reset_4 := FALSE;
   END_IF;
END_REGION

REGION Network 5: Increase Counter-1 (and convert sec to hour)
   IF #IN THEN #Accum_1 := #Accum_1 + 5; END_IF;
   #Cnt_Hours_1 := #Accum_1 / 3600;
   #tmp_bool := #IN;
END_REGION

REGION Network 6: Increase Counter-2 (and convert sec to hour)
   IF #IN THEN #Accum_2 := #Accum_2 + 5; END_IF;
   #Cnt_Hours_2 := #Accum_2 / 3600;
   #tmp_bool := #IN;
END_REGION

REGION Network 7: Increase Counter-3 (and convert sec to hour)
   IF #IN THEN #Accum_3 := #Accum_3 + 5; END_IF;
   #Cnt_Hours_3 := #Accum_3 / 3600;
   #tmp_bool := #IN;
END_REGION

REGION Network 8: Increase Counter-4 (and convert sec to hour)
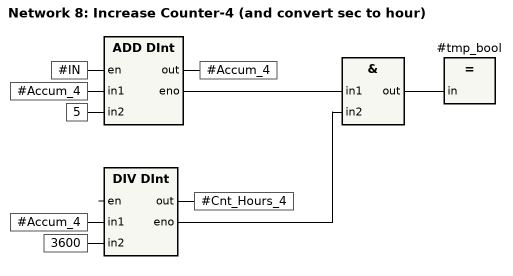
   IF #IN THEN #Accum_4 := #Accum_4 + 5; END_IF;
   #Cnt_Hours_4 := #Accum_4 / 3600;
   #tmp_bool := #IN;
END_REGION
END_FUNCTION_BLOCK

FUNCTION_BLOCK "ACESYS_MASTER"   // FB200, FBD
TITLE = ACESYS V8.0 - Build 001 - MASTER Block
{ S7_Optimized_Access := 'FALSE' }
AUTHOR : FLSmidth
FAMILY : ACESYS
NAME : MASTER
VERSION : 8.0
   VAR_INPUT
      LOC_TYPE : Bool;   // Accept return in local without command: "0"= Disable / "1" = Enable
      REM_TYPE : Bool;   // REM Switch Type : "0"= Normal / "1" = Force Local
      SIM_ENABLE : Bool;   // Enable Device Simulation : "0"= Disable / "1" = Enable
      SS_FP_ENABLE : Bool := TRUE;   // Enable Single Start from FP : "0"= Disable / "1" = Enable
      SS_Field_ENABLE : Bool := TRUE;   // Enable Single Start from Field: "0"= Disable / "1" = Enable
      MAN_ENABLE : Bool := TRUE;   // Enable Manual Mode : "0"= Disable / "1" = Enable
      LOC_ENABLE : Bool := TRUE;   // Enable Manual Local : "0"= Disable / "1" = Enable
      TEST_ENABLE : Bool := TRUE;   // Enable Test Mode : "0"= Disable / "1" = Enable
      QSTOP_FP_Unit : Bool;   // Enable Quick Stop from Unit FP: "0"= Disable / "1" = Enable
      RED_ENABLE : Bool;   // Redundant system : "0"= Disable / "1" = Enable
      WatchDog_HMI_Enable : Bool;   // Enable Watchdog Supervision : "0"= Disable / "1" = Enable
      WatchDog_HMI_Time : Time := T#30MS;   // WatchDog Time HMI
      OB1_CycleTime : Int;
   END_VAR
   VAR_OUTPUT
      WatchDog_HMI_Elap : Time;   // WatchDog HMI Elapsed Time
      MASTER_Link : "ACESYS_MASTER_LINK";   // Link to Departments
      First_Scan : Bool;   // First Scan Pulse
      SEC_Toggle : Bool;   // 1 Sec. Toggle
   END_VAR
   VAR_IN_OUT
      WatchDog_HMI : Bool;   // WatchDog Pulse from HMI
   END_VAR
   VAR
      BlockInfo : Struct
         Ace_Version : Int;   // Acesys Block Version Number
         Ace_BuildNo : Int;   // Acesys Block Build Number
         State_Act : Int;   // Actual State Number
         State_Prev : Int;   // Previous State Number
         DB_Number : Int;   // Block Instance DB Number
      END_STRUCT;
      SZL : Struct
         Lenghtdr : Word;   // Lenght data-area
         N_DR : Word;   // Number of in data-area
      END_STRUCT;
      DR : Struct
         RedInfo : Word;   // Info on redundancy W#16#0011: Single H CPU / W#16#0012: 1 of 2 H system
         Reserved_Bit_0 : Bool;   // mwstat1 / Reserved
         Reserved_Bit_1 : Bool;   // mwstat1 / Reserved
         Reserved_Bit_2 : Bool;   // mwstat1 / Reserved
         Reserved_Bit_3 : Bool;   // mwstat1 / Reserved
         H_Status_Rack0_Master : Bool;   // H status of CPU in Rack 0 =0: Standby CPU / =1:master CPU
         H_Status_Rack1_Master : Bool;   // H status of CPU in Rack 1 =0: Standby CPU / =1:master CPU
         Reserved_Bit_6 : Bool;   // mwstat1 / Reserved
         Reserved_Bit_7 : Bool;   // mwstat1 / Reserved
         MwStat2 : Byte;   // Status byte2
         hsfcinfo : Word;   // Info word on SFC 90
         CommonError : Word;   // Group error word
         Bz_CPU0 : Word;   // Operating status CPU 0
         Bz_CPU1 : Word;   // Operating status CPU 1
         Bz_CPU2 : Word;   // Reserved
         Cpu_valid : Byte;   // Validity of variables
         Reserve : Byte;   // Reserved
      END_STRUCT;
      Timer_Watchdog : TON_TIME;
      TimerSlow_On : TON_TIME;
      TimerSlow_Off : TON_TIME;
      TimerFast_On : TON_TIME;
      TimerFast_Off : TON_TIME;
      Flash_Slow : Bool;
      Flash_Fast : Bool;
      FirstScan : Bool;
      FirstScan_Hlp : Bool;
      Clock_Sec_Old : USInt;
      Clock_Min_Old : USInt;
      Clock_Hour_Old : USInt;
      Clock_Day_Old : USInt;
      Clock_Month_Old : USInt;
      Clock_Year_Old : UInt;
      Toggle : Bool;
      Master_Link_Internal : "ACESYS_MASTER_LINK";
   END_VAR
   VAR_TEMP
      AOn : Bool;   // Always On
      AOff : Bool;   // Always Off
      TimeOut : Bool;
      Set : Bool;
      Reset : Bool;
      DummyBool : Bool;
      Busy : Bool;
      TimerOut : Bool;
      RETVAL : Int;
      TempDINT : DInt;
      Clock_Sec : USInt;
      Clock_Min : USInt;
      Clock_Hour : USInt;
      Clock_Day : USInt;
      Clock_Month : USInt;
      Clock_Year : UInt;
      SysTime : DTL;
      Actual_Time : Time_Of_Day;
   END_VAR
   VAR_TEMP   // added for the SCL form of the ladder/FBD networks
      _w1 : Bool;
   END_VAR
BEGIN

REGION Network 1: Always On/Off
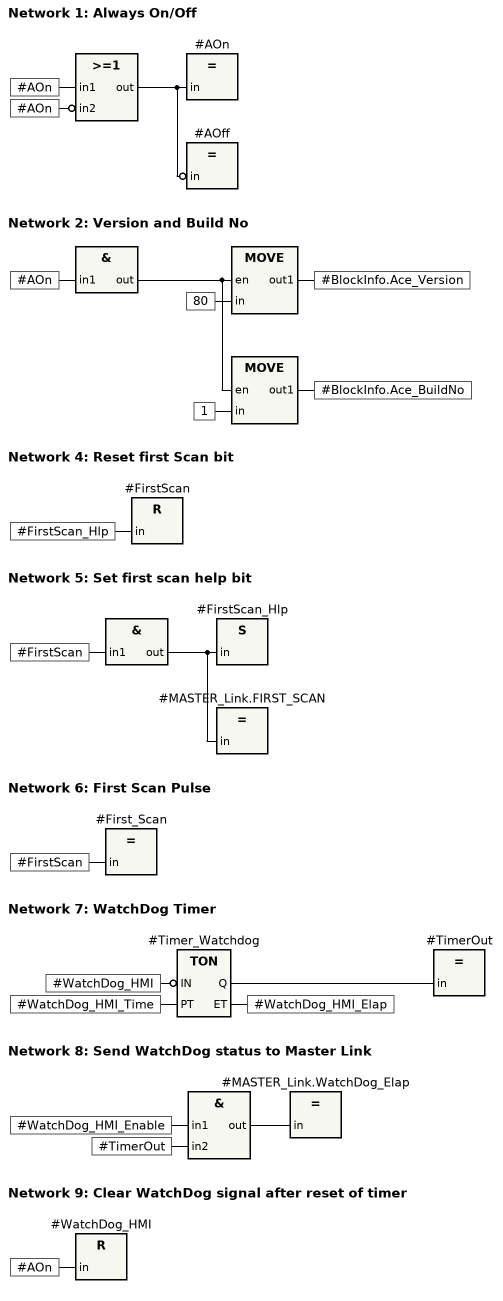
   #AOn := #AOn OR NOT #AOn;
   #AOff := NOT #AOn;
END_REGION

REGION Network 2: Version and Build No
   IF #AOn THEN
       #BlockInfo.Ace_Version := 80;
       #BlockInfo.Ace_BuildNo := 1;
   END_IF;
END_REGION

REGION Network 3 (STL): Instance DB Number to Faceplate
         L     DINO;
         T     #BlockInfo.DB_Number;
END_REGION

REGION Network 4: Reset first Scan bit
   IF #FirstScan_Hlp THEN #FirstScan := FALSE; END_IF;
END_REGION

REGION Network 5: Set first scan help bit
   IF #FirstScan THEN #FirstScan_Hlp := TRUE; END_IF;
   #MASTER_Link.FIRST_SCAN := #FirstScan;
END_REGION

REGION Network 6: First Scan Pulse
   #First_Scan := #FirstScan;
END_REGION

REGION Network 7: WatchDog Timer
   #Timer_Watchdog(IN := NOT #WatchDog_HMI, PT := #WatchDog_HMI_Time, ET => #WatchDog_HMI_Elap);   // TON
   #TimerOut := #Timer_Watchdog.Q;
END_REGION

REGION Network 8: Send WatchDog status to Master Link
   #MASTER_Link.WatchDog_Elap := #WatchDog_HMI_Enable AND #TimerOut;
END_REGION

REGION Network 9: Clear WatchDog signal after reset of timer
   IF #AOn THEN #WatchDog_HMI := FALSE; END_IF;
END_REGION

REGION Network 10
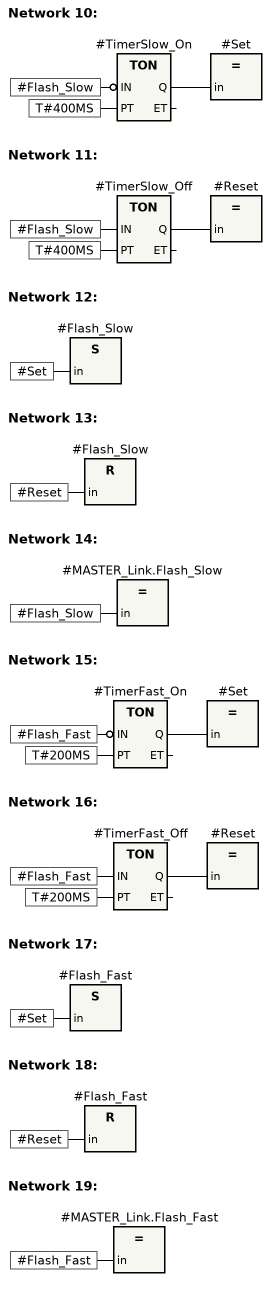
   #TimerSlow_On(IN := NOT #Flash_Slow, PT := T#400MS);   // TON
   #Set := #TimerSlow_On.Q;
END_REGION

REGION Network 11
   #TimerSlow_Off(IN := #Flash_Slow, PT := T#400MS);   // TON
   #Reset := #TimerSlow_Off.Q;
END_REGION

REGION Network 12
   IF #Set THEN #Flash_Slow := TRUE; END_IF;
END_REGION

REGION Network 13
   IF #Reset THEN #Flash_Slow := FALSE; END_IF;
END_REGION

REGION Network 14
   #MASTER_Link.Flash_Slow := #Flash_Slow;
END_REGION

REGION Network 15
   #TimerFast_On(IN := NOT #Flash_Fast, PT := T#200MS);   // TON
   #Set := #TimerFast_On.Q;
END_REGION

REGION Network 16
   #TimerFast_Off(IN := #Flash_Fast, PT := T#200MS);   // TON
   #Reset := #TimerFast_Off.Q;
END_REGION

REGION Network 17
   IF #Set THEN #Flash_Fast := TRUE; END_IF;
END_REGION

REGION Network 18
   IF #Reset THEN #Flash_Fast := FALSE; END_IF;
END_REGION

REGION Network 19
   #MASTER_Link.Flash_Fast := #Flash_Fast;
END_REGION

REGION Network 20: Read PLC time
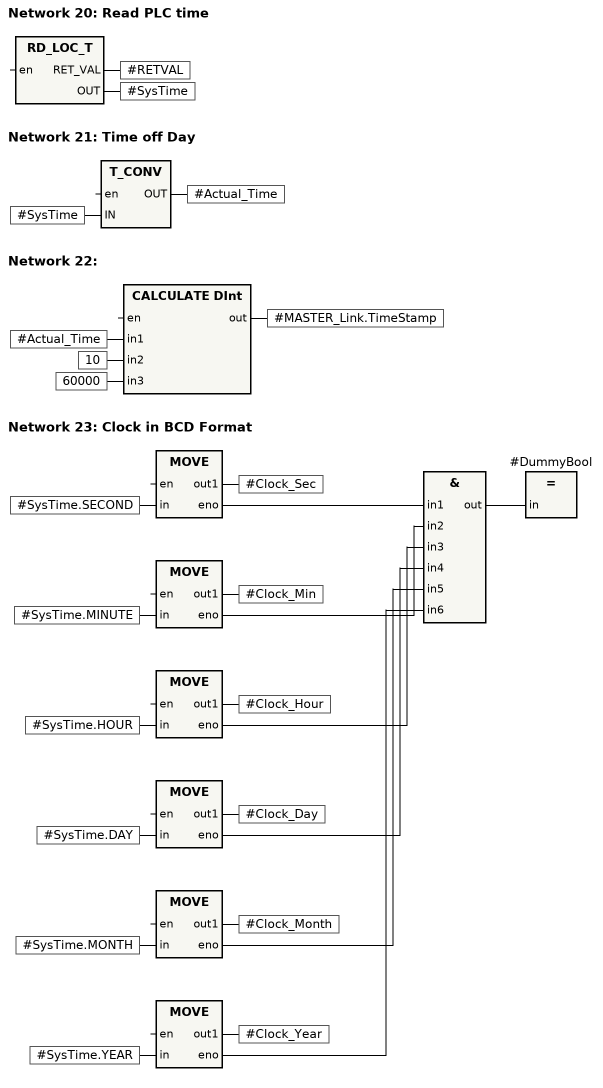
   #RETVAL := RD_LOC_T(OUT => #SysTime);
END_REGION

REGION Network 21: Time off Day
   #Actual_Time := T_CONV(IN := #SysTime);
END_REGION

REGION Network 22
   // Modolus calculation
   // Actual time = 00:00:00 -> 0000000ms  12:00:00 -> 4300000ms
   // 
   // Time Stamp =
   // (Min 0-9*60*100+Msec*0.1)  -> Actual time/10 MOD 60000
   #MASTER_Link.TimeStamp := (#Actual_Time/10)MOD 60000;
END_REGION

REGION Network 23: Clock in BCD Format
   #Clock_Sec := #SysTime.SECOND;
   #Clock_Min := #SysTime.MINUTE;
   #Clock_Hour := #SysTime.HOUR;
   #Clock_Day := #SysTime.DAY;
   #Clock_Month := #SysTime.MONTH;
   #Clock_Year := #SysTime.YEAR;
   #DummyBool := TRUE;
END_REGION

REGION Network 24: Pulse per Second
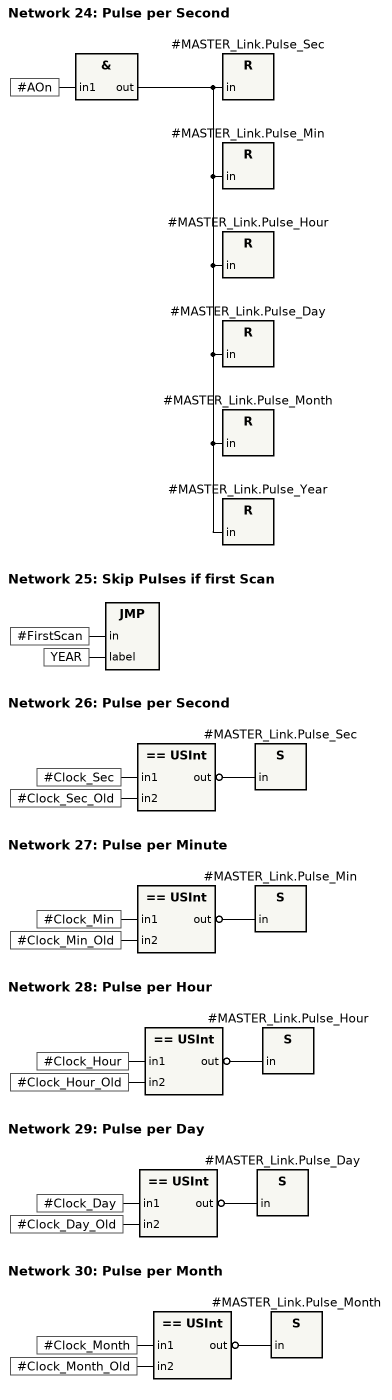
   IF #AOn THEN
       #MASTER_Link.Pulse_Sec := FALSE;
       #MASTER_Link.Pulse_Min := FALSE;
       #MASTER_Link.Pulse_Hour := FALSE;
       #MASTER_Link.Pulse_Day := FALSE;
       #MASTER_Link.Pulse_Month := FALSE;
       #MASTER_Link.Pulse_Year := FALSE;
   END_IF;
END_REGION

REGION Network 25: Skip Pulses if first Scan
   IF #FirstScan THEN GOTO YEAR; END_IF;
END_REGION

REGION Network 26: Pulse per Second
   IF NOT (#Clock_Sec = #Clock_Sec_Old) THEN #MASTER_Link.Pulse_Sec := TRUE; END_IF;
END_REGION

REGION Network 27: Pulse per Minute
   IF NOT (#Clock_Min = #Clock_Min_Old) THEN #MASTER_Link.Pulse_Min := TRUE; END_IF;
END_REGION

REGION Network 28: Pulse per Hour
   IF NOT (#Clock_Hour = #Clock_Hour_Old) THEN #MASTER_Link.Pulse_Hour := TRUE; END_IF;
END_REGION

REGION Network 29: Pulse per Day
   IF NOT (#Clock_Day = #Clock_Day_Old) THEN #MASTER_Link.Pulse_Day := TRUE; END_IF;
END_REGION

REGION Network 30: Pulse per Month
   IF NOT (#Clock_Month = #Clock_Month_Old) THEN #MASTER_Link.Pulse_Month := TRUE; END_IF;
END_REGION

REGION Network 31: Pulse per Year
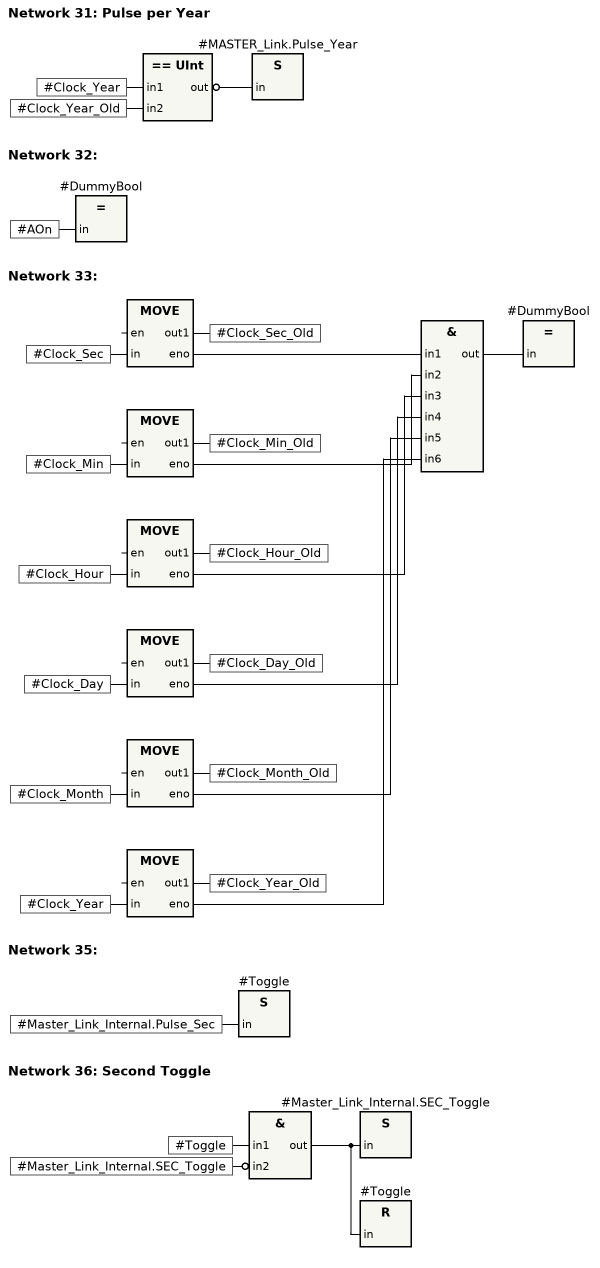
   IF NOT (#Clock_Year = #Clock_Year_Old) THEN #MASTER_Link.Pulse_Year := TRUE; END_IF;
END_REGION

REGION Network 32
   YEAR:
   #DummyBool := #AOn;
END_REGION

REGION Network 33
   #Clock_Sec_Old := #Clock_Sec;
   #Clock_Min_Old := #Clock_Min;
   #Clock_Hour_Old := #Clock_Hour;
   #Clock_Day_Old := #Clock_Day;
   #Clock_Month_Old := #Clock_Month;
   #Clock_Year_Old := #Clock_Year;
   #DummyBool := TRUE;
END_REGION

REGION Network 34 (SCL): Copy Master Link Variables to Stat - Indirect
   #Master_Link_Internal.Pulse_Sec := PEEK_BOOL(area := 16#84, dbNumber := #BlockInfo.DB_Number, byteOffset := 12, bitOffset := 2);
   #Master_Link_Internal.SEC_Toggle := PEEK_BOOL(area := 16#84, dbNumber := #BlockInfo.DB_Number, byteOffset := 14, bitOffset := 3);
END_REGION

REGION Network 35
   IF #Master_Link_Internal.Pulse_Sec THEN #Toggle := TRUE; END_IF;
END_REGION

REGION Network 36: Second Toggle
   #_w1 := #Toggle AND NOT #Master_Link_Internal.SEC_Toggle;
   IF #_w1 THEN
       #Master_Link_Internal.SEC_Toggle := TRUE;
       #Toggle := FALSE;
   END_IF;
END_REGION

REGION Network 37: Second Toggle
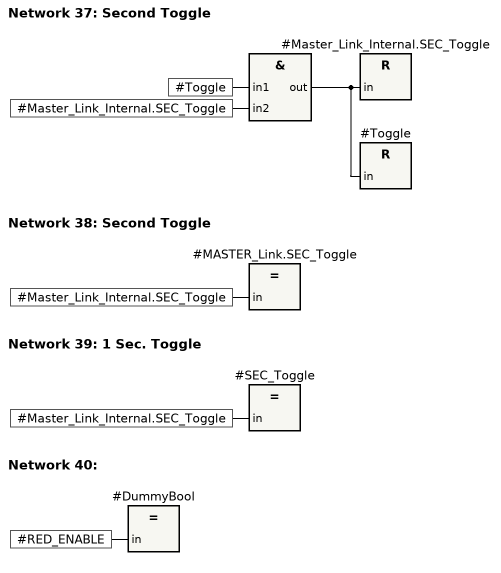
   #_w1 := #Toggle AND #Master_Link_Internal.SEC_Toggle;
   IF #_w1 THEN
       #Master_Link_Internal.SEC_Toggle := FALSE;
       #Toggle := FALSE;
   END_IF;
END_REGION

REGION Network 38: Second Toggle
   #MASTER_Link.SEC_Toggle := #Master_Link_Internal.SEC_Toggle;
END_REGION

REGION Network 39: 1 Sec. Toggle
   #SEC_Toggle := #Master_Link_Internal.SEC_Toggle;
END_REGION

REGION Network 40
   // Redundancy not supported yet in 1500 series, Redundancy status check blocks removed
   #DummyBool := #RED_ENABLE;
END_REGION

REGION Network 41: Device Simulation Enabled
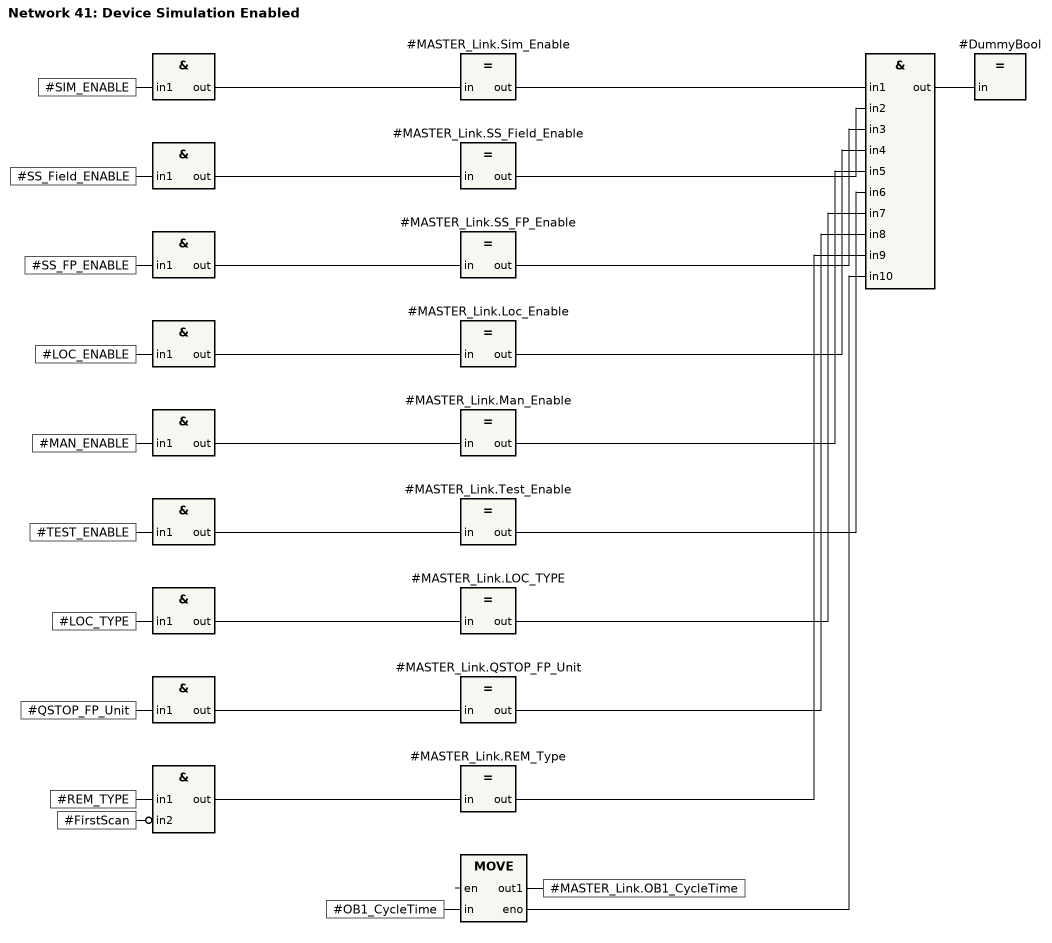
   #MASTER_Link.Sim_Enable := #SIM_ENABLE;
   #MASTER_Link.SS_Field_Enable := #SS_Field_ENABLE;
   #MASTER_Link.SS_FP_Enable := #SS_FP_ENABLE;
   #MASTER_Link.Loc_Enable := #LOC_ENABLE;
   #MASTER_Link.Man_Enable := #MAN_ENABLE;
   #MASTER_Link.Test_Enable := #TEST_ENABLE;
   #MASTER_Link.LOC_TYPE := #LOC_TYPE;
   #MASTER_Link.QSTOP_FP_Unit := #QSTOP_FP_Unit;
   #MASTER_Link.REM_Type := #REM_TYPE AND NOT #FirstScan;
   #MASTER_Link.OB1_CycleTime := #OB1_CycleTime;
   #DummyBool := #SIM_ENABLE AND #SS_Field_ENABLE AND #SS_FP_ENABLE AND #LOC_ENABLE AND #MAN_ENABLE AND #TEST_ENABLE AND #LOC_TYPE AND #QSTOP_FP_Unit AND #MASTER_Link.REM_Type;
END_REGION
END_FUNCTION_BLOCK

FUNCTION_BLOCK "ACESYS_DEPT"   // FB201, FBD
TITLE = ACESYS V8.0 - Build 001 - DEPARTMENT Block
{ S7_Optimized_Access := 'FALSE' }
AUTHOR : FLSmidth
FAMILY : ACESYS
NAME : DEPT
VERSION : 8.0
   VAR_INPUT
      Master_Link : "ACESYS_MASTER_LINK";
      EnCtrl : Bool;   // Enable Faceplate Control
      DEMER : Bool;   // Department Emergency Stop
      START : Bool;   // Department Start
      STOP : Bool;   // Department Stop
      RST : Bool;   // Department Reset
   END_VAR
   VAR_OUTPUT
      DEPT_LINK : "ACESYS_DEPT_LINK";   // Acesys Department Commands
      MSW : "ACESYS_HMI_STAT_32T";
   END_VAR
   VAR
      BlockInfo : Struct
         Ace_Version : Int;   // Acesys Block Version Number
         Ace_BuildNo : Int;   // Acesys Block Build Number
         DB_Number : Int;   // Block Instance DB Number
      END_STRUCT;
      FP_CMD : Struct   // Faceplate Commands
         Spare_08 : Bool;
         Spare_09 : Bool;
         Spare_10 : Bool;
         Spare_11 : Bool;
         SelAndStart : Bool;
         DeselAndStop : Bool;
         Spare_14 : Bool;
         AckAlarm : Bool;
         Select : Bool;
         Deselect : Bool;
         Start : Bool;
         Stop : Bool;
         MasterStop : Bool;
         QuickStop : Bool;
         Spare_06 : Bool;
         Spare_07 : Bool;
      END_STRUCT;
      FP_DIM : Struct   // Faceplate Dimmed Buttons
         Select : Bool;   // DimOut
         DeSelect : Bool;   // DimOut
         Start : Bool;   // DimOut
         Stop : Bool;   // DimOut
         QuickStop : Bool;   // DimOut
         MasterStop : Bool;   // DimOut
      END_STRUCT;
      START_Int : Bool;   // Internal Start Bit
      Stop_int : Bool;   // Internal Stop Bit
      DEP_Sel_Int : Bool;   // Internal Department Select Bit
      Dep_DeSel_Int : Bool;   // Internal Department DeSelect Bit
      Selecting : Bool;
      Deselecting : Bool;
      ONS_Start : Bool;   // OneShot bit
      ONS_FS_Reset : Bool;   // OneShot bit
      ONS_RST : Bool;   // OneShot bit
      MSW_Status : Int;   // Internal Status Word
      StatusToECS : Int;   // Temp Status
      Dept_Link_Internal : "ACESYS_DEPT_LINK";   // Internal Dept Link for block logic
      MSW_Status_Trans : Int;   // Transfer MSW Status
   END_VAR
   VAR_TEMP
      AOn : Bool;   // Always On
      AOff : Bool;   // Always Off
      DummyBool : Bool;
      ECSStatusBuilder : Int;   // Temp Status
   END_VAR
   VAR_TEMP   // added for the SCL form of the ladder/FBD networks
      _w1 : Bool;
      _w2 : Bool;
   END_VAR
BEGIN

REGION Network 1: Always On
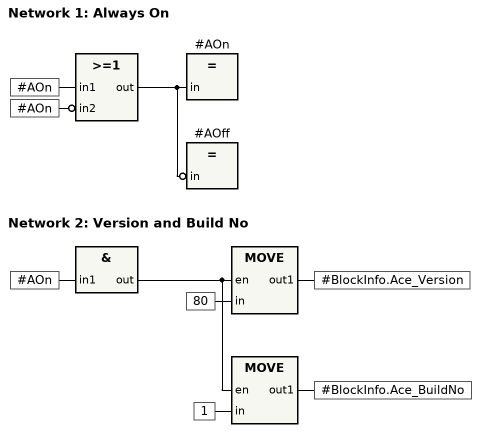
   #AOn := #AOn OR NOT #AOn;
   #AOff := NOT #AOn;
END_REGION

REGION Network 2: Version and Build No
   IF #AOn THEN
       #BlockInfo.Ace_Version := 80;
       #BlockInfo.Ace_BuildNo := 1;
   END_IF;
END_REGION

REGION Network 3 (STL): Instance DB Number to Faceplate
         L     DINO;
         T     #BlockInfo.DB_Number;
END_REGION

REGION Network 4 (SCL): Transfer Actual Dept Link to Depaetment Link Internal
   #Dept_Link_Internal.Reset := PEEK_BOOL(area := 16#84, dbNumber := #BlockInfo.DB_Number, byteOffset := 14, bitOffset := 0);
   #Dept_Link_Internal.Start := PEEK_BOOL(area := 16#84, dbNumber := #BlockInfo.DB_Number, byteOffset := 14, bitOffset := 1);
   #Dept_Link_Internal.Stop := PEEK_BOOL(area := 16#84, dbNumber := #BlockInfo.DB_Number, byteOffset := 14, bitOffset := 2);
   #Dept_Link_Internal.MasterStop := PEEK_BOOL(area := 16#84, dbNumber := #BlockInfo.DB_Number, byteOffset := 14, bitOffset := 3);
   #Dept_Link_Internal.QuickStop := PEEK_BOOL(area := 16#84, dbNumber := #BlockInfo.DB_Number, byteOffset := 14, bitOffset := 4);
   #Dept_Link_Internal.DeptSelect := PEEK_BOOL(area := 16#84, dbNumber := #BlockInfo.DB_Number, byteOffset := 14, bitOffset := 5);
   #Dept_Link_Internal.DeptDeSelect := PEEK_BOOL(area := 16#84, dbNumber := #BlockInfo.DB_Number, byteOffset := 14, bitOffset := 6);
   #Dept_Link_Internal.All_Group_ON := PEEK_BOOL(area := 16#84, dbNumber := #BlockInfo.DB_Number, byteOffset := 17, bitOffset := 0);
   #Dept_Link_Internal.All_Group_OFF := PEEK_BOOL(area := 16#84, dbNumber := #BlockInfo.DB_Number, byteOffset := 17, bitOffset := 1);
   #Dept_Link_Internal.All_Group_Sel_RDY := PEEK_BOOL(area := 16#84, dbNumber := #BlockInfo.DB_Number, byteOffset := 17, bitOffset := 2);
   #Dept_Link_Internal.All_Selected := PEEK_BOOL(area := 16#84, dbNumber := #BlockInfo.DB_Number, byteOffset := 17, bitOffset := 3);
   #Dept_Link_Internal.All_DeSelected := PEEK_BOOL(area := 16#84, dbNumber := #BlockInfo.DB_Number, byteOffset := 17, bitOffset := 4);
   #Dept_Link_Internal.All_Selected_Running := PEEK_BOOL(area := 16#84, dbNumber := #BlockInfo.DB_Number, byteOffset := 17, bitOffset := 5);
   #Dept_Link_Internal.Ready_For_StopCmd := PEEK_BOOL(area := 16#84, dbNumber := #BlockInfo.DB_Number, byteOffset := 17, bitOffset := 6);
   #Dept_Link_Internal.WatchDog_Failure := PEEK_BOOL(area := 16#84, dbNumber := #BlockInfo.DB_Number, byteOffset := 17, bitOffset := 7);
END_REGION

REGION Network 5: DimOut
   // >>>>> DIM Push Buttons on Faceplate <<<<<
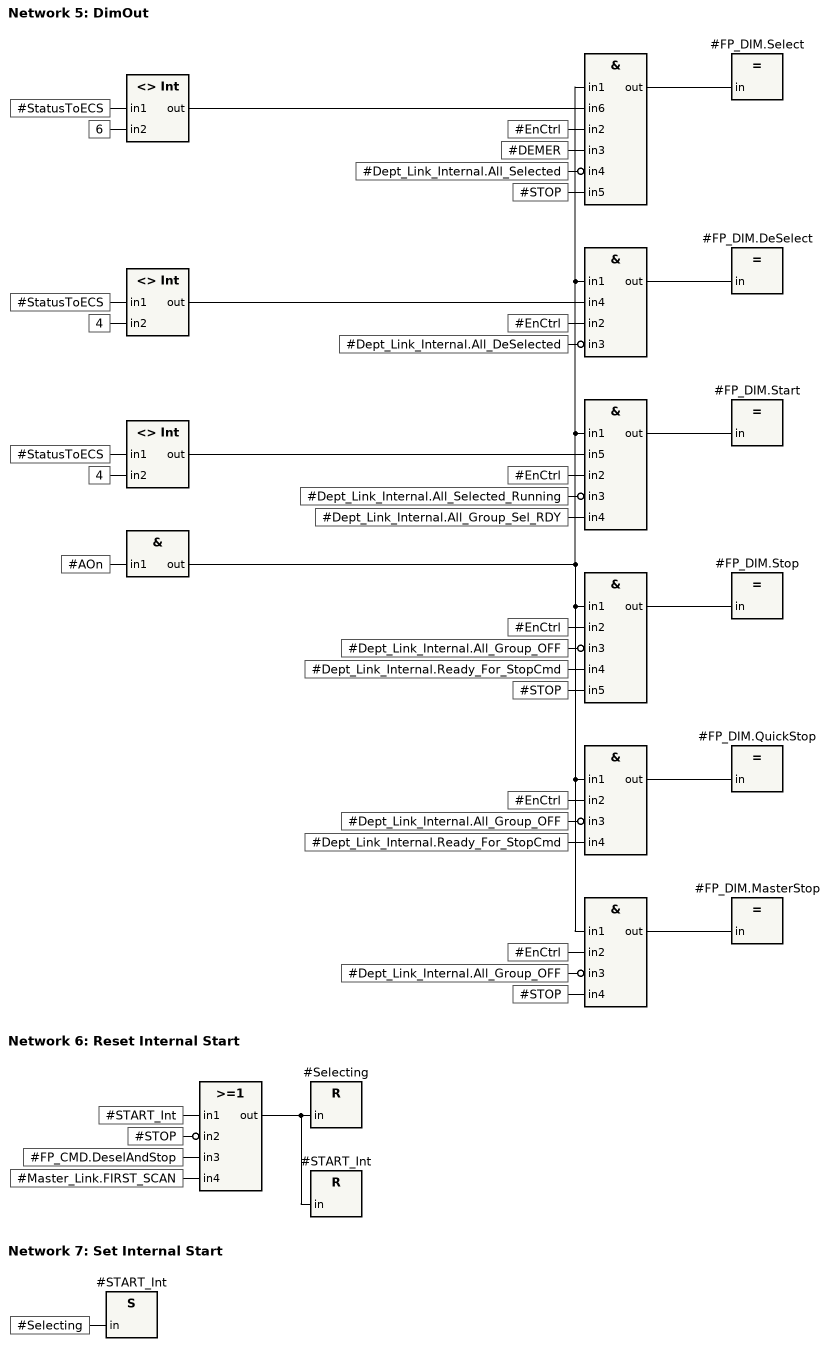
   #FP_DIM.Select := #AOn AND (#StatusToECS <> 6) AND #EnCtrl AND #DEMER AND NOT #Dept_Link_Internal.All_Selected AND #STOP;
   #FP_DIM.DeSelect := #AOn AND (#StatusToECS <> 4) AND #EnCtrl AND NOT #Dept_Link_Internal.All_DeSelected;
   #FP_DIM.Start := #AOn AND (#StatusToECS <> 4) AND #EnCtrl AND NOT #Dept_Link_Internal.All_Selected_Running AND #Dept_Link_Internal.All_Group_Sel_RDY;
   #FP_DIM.Stop := #AOn AND #EnCtrl AND NOT #Dept_Link_Internal.All_Group_OFF AND #Dept_Link_Internal.Ready_For_StopCmd AND #STOP;
   #FP_DIM.QuickStop := #AOn AND #EnCtrl AND NOT #Dept_Link_Internal.All_Group_OFF AND #Dept_Link_Internal.Ready_For_StopCmd;
   #FP_DIM.MasterStop := #AOn AND #EnCtrl AND NOT #Dept_Link_Internal.All_Group_OFF AND #STOP;
END_REGION

REGION Network 6: Reset Internal Start
   IF #START_Int OR NOT #STOP OR #FP_CMD.DeselAndStop OR #Master_Link.FIRST_SCAN THEN
       #Selecting := FALSE;
       #START_Int := FALSE;
   END_IF;
END_REGION

REGION Network 7: Set Internal Start
   IF #Selecting THEN #START_Int := TRUE; END_IF;
END_REGION

REGION Network 8: Selecting Groups
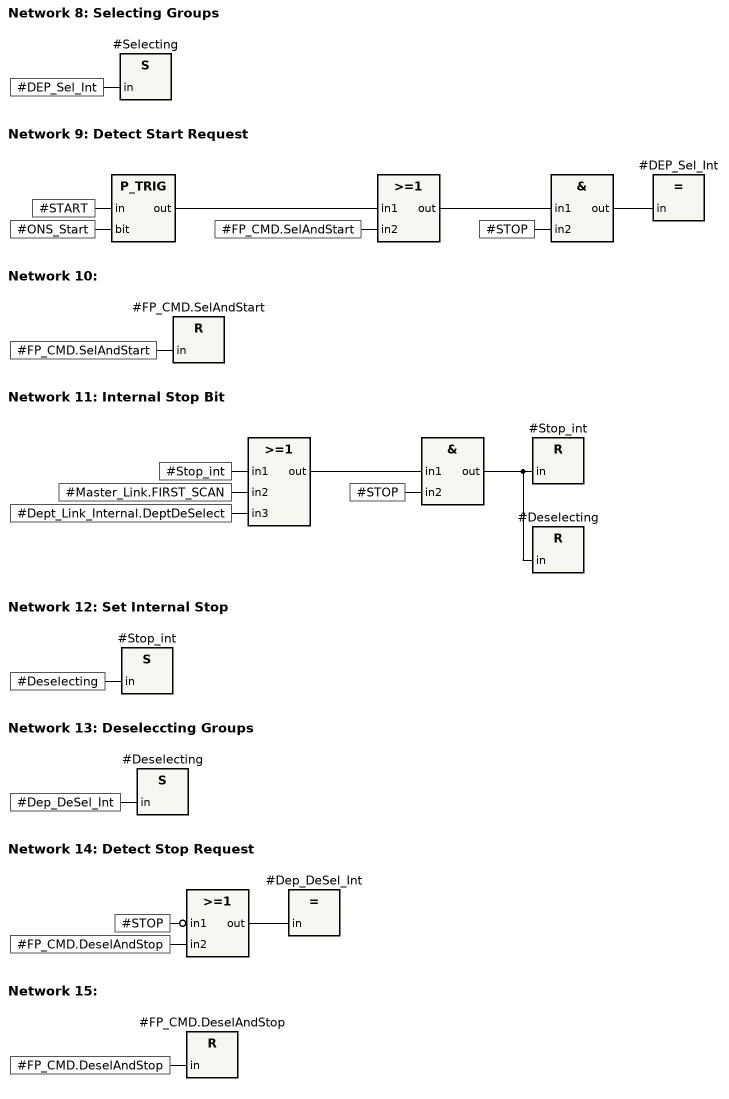
   IF #DEP_Sel_Int THEN #Selecting := TRUE; END_IF;
END_REGION

REGION Network 9: Detect Start Request
   #_w1 := #START AND NOT #ONS_Start;   // rising edge
   #ONS_Start := #START;
   #DEP_Sel_Int := (#_w1 OR #FP_CMD.SelAndStart) AND #STOP;
END_REGION

REGION Network 10
   IF #FP_CMD.SelAndStart THEN #FP_CMD.SelAndStart := FALSE; END_IF;
END_REGION

REGION Network 11: Internal Stop Bit
   #_w1 := (#Stop_int OR #Master_Link.FIRST_SCAN OR #Dept_Link_Internal.DeptDeSelect) AND #STOP;
   IF #_w1 THEN
       #Stop_int := FALSE;
       #Deselecting := FALSE;
   END_IF;
END_REGION

REGION Network 12: Set Internal Stop
   IF #Deselecting THEN #Stop_int := TRUE; END_IF;
END_REGION

REGION Network 13: Deseleccting Groups
   IF #Dep_DeSel_Int THEN #Deselecting := TRUE; END_IF;
END_REGION

REGION Network 14: Detect Stop Request
   #Dep_DeSel_Int := NOT #STOP OR #FP_CMD.DeselAndStop;
END_REGION

REGION Network 15
   IF #FP_CMD.DeselAndStop THEN #FP_CMD.DeselAndStop := FALSE; END_IF;
END_REGION

REGION Network 16: Alarm Reset
   // >>>>> FACEPLATE COMMANDS (Pulse Type) <<<<<
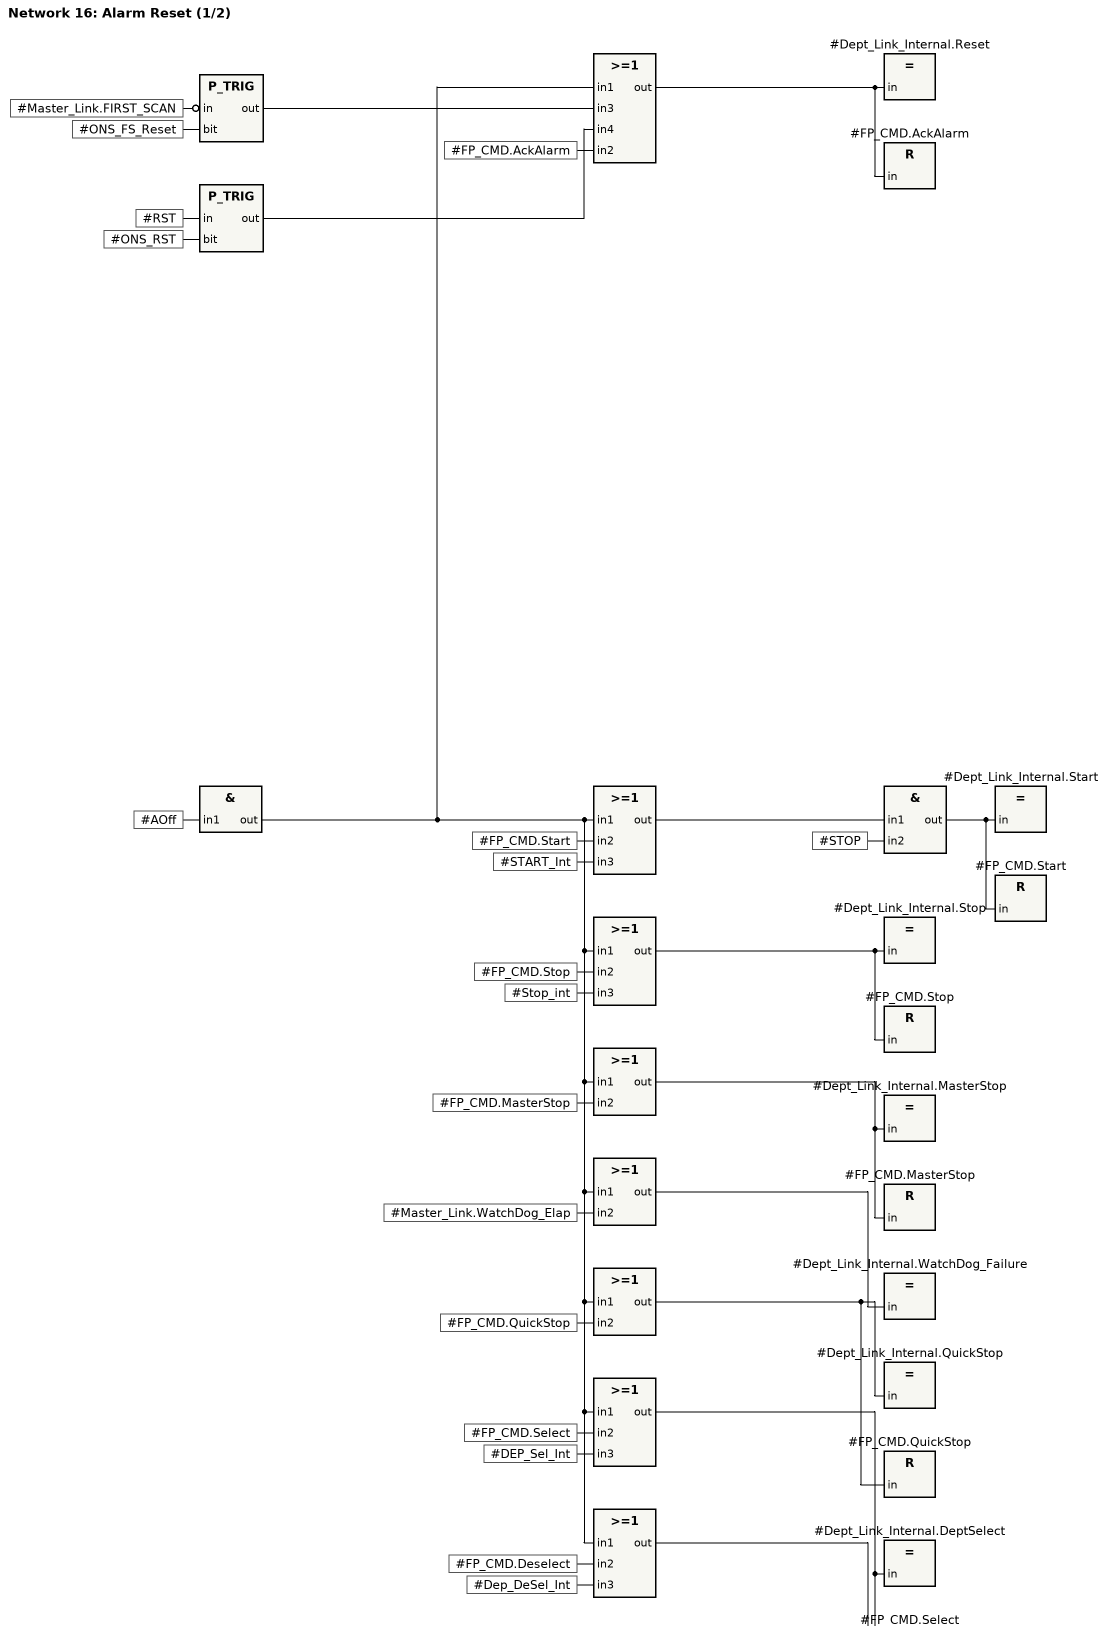
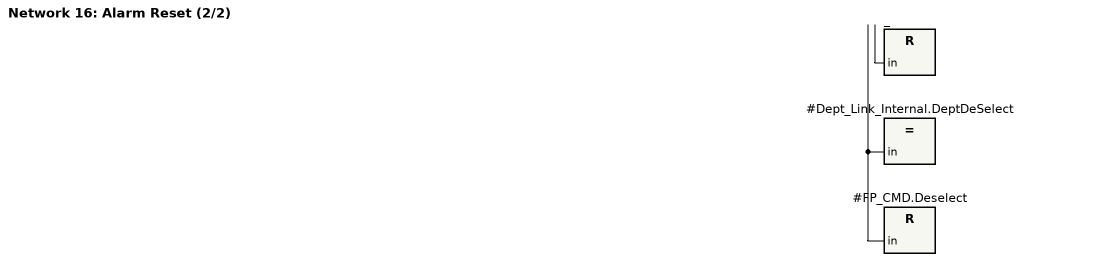
   #_w1 := NOT #Master_Link.FIRST_SCAN AND NOT #ONS_FS_Reset;   // rising edge
   #ONS_FS_Reset := NOT #Master_Link.FIRST_SCAN;
   #_w2 := #RST AND NOT #ONS_RST;   // rising edge
   #ONS_RST := #RST;
   #Dept_Link_Internal.Reset := #AOff OR #_w1 OR #_w2 OR #FP_CMD.AckAlarm;
   IF #Dept_Link_Internal.Reset THEN #FP_CMD.AckAlarm := FALSE; END_IF;
   #Dept_Link_Internal.Start := (#AOff OR #FP_CMD.Start OR #START_Int) AND #STOP;
   IF #Dept_Link_Internal.Start THEN #FP_CMD.Start := FALSE; END_IF;
   #Dept_Link_Internal.Stop := #AOff OR #FP_CMD.Stop OR #Stop_int;
   IF #Dept_Link_Internal.Stop THEN #FP_CMD.Stop := FALSE; END_IF;
   #Dept_Link_Internal.MasterStop := #AOff OR #FP_CMD.MasterStop;
   IF #Dept_Link_Internal.MasterStop THEN #FP_CMD.MasterStop := FALSE; END_IF;
   #Dept_Link_Internal.WatchDog_Failure := #AOff OR #Master_Link.WatchDog_Elap;
   #Dept_Link_Internal.QuickStop := #AOff OR #FP_CMD.QuickStop;
   IF #Dept_Link_Internal.QuickStop THEN #FP_CMD.QuickStop := FALSE; END_IF;
   #Dept_Link_Internal.DeptSelect := #AOff OR #FP_CMD.Select OR #DEP_Sel_Int;
   IF #Dept_Link_Internal.DeptSelect THEN #FP_CMD.Select := FALSE; END_IF;
   #Dept_Link_Internal.DeptDeSelect := #AOff OR #FP_CMD.Deselect OR #Dep_DeSel_Int;
   IF #Dept_Link_Internal.DeptDeSelect THEN #FP_CMD.Deselect := FALSE; END_IF;
END_REGION

REGION Network 17: Pass Time Stamp
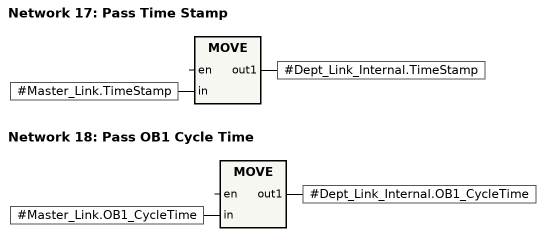
   #Dept_Link_Internal.TimeStamp := #Master_Link.TimeStamp;
END_REGION

REGION Network 18: Pass OB1 Cycle Time
   #Dept_Link_Internal.OB1_CycleTime := #Master_Link.OB1_CycleTime;
END_REGION

REGION Network 19: Status to ECS
   // 1 = All Stopped
   // 2 = All Running
   // 3 = External Started
   // 4 = Master Stopping
   // 5 = Watch Dog Stopping
   // 6 = Quick Stop
   // 7 = Aelected to Start
   // 8 = Stop Active from user Program
   // 
   // 200 = Department Emergency stop
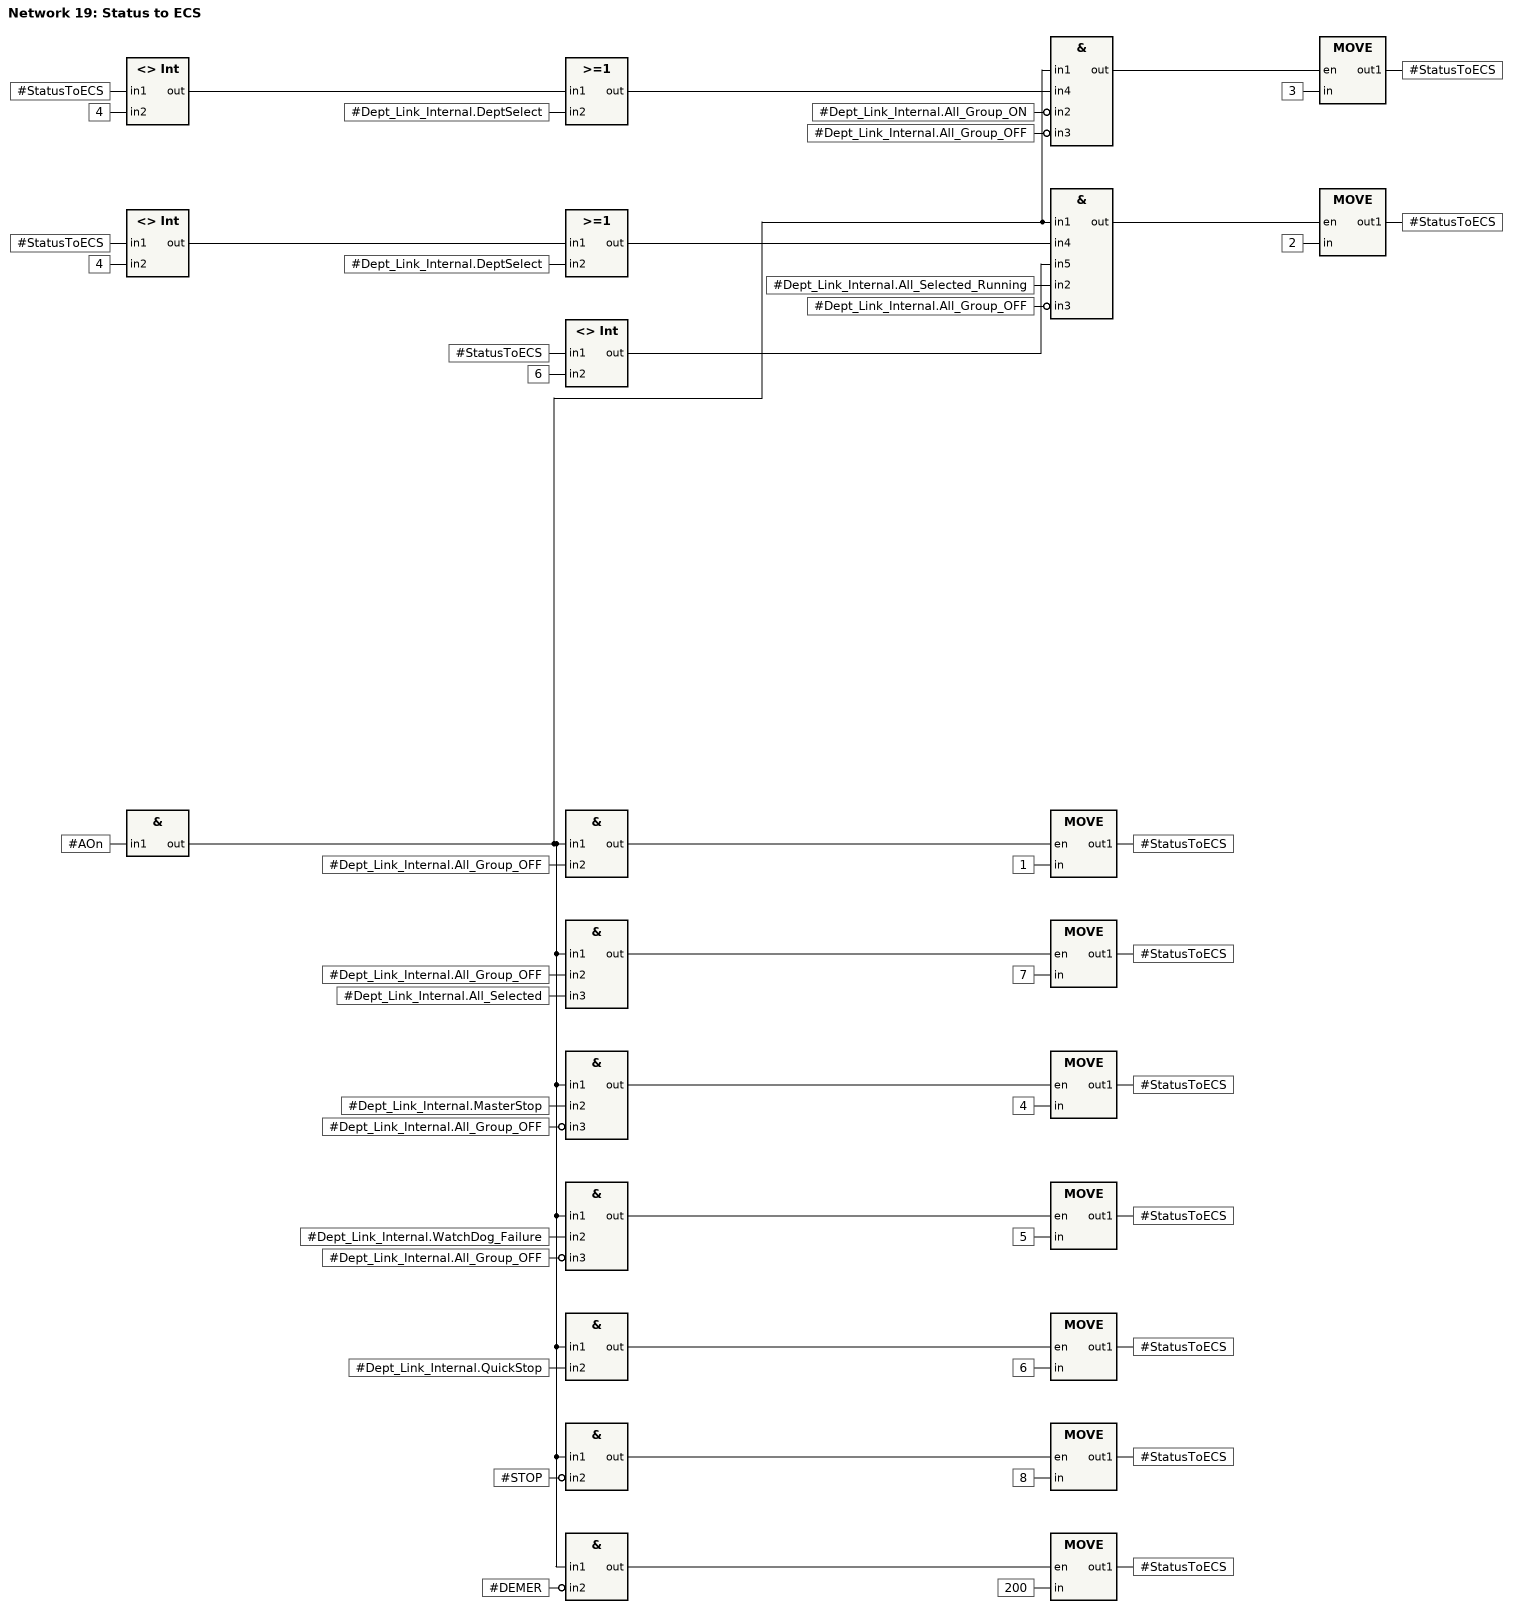
   IF #AOn AND ((#StatusToECS <> 4) OR #Dept_Link_Internal.DeptSelect) AND NOT #Dept_Link_Internal.All_Group_ON AND NOT #Dept_Link_Internal.All_Group_OFF THEN
       #StatusToECS := 3;
   END_IF;
   IF #AOn AND ((#StatusToECS <> 4) OR #Dept_Link_Internal.DeptSelect) AND (#StatusToECS <> 6) AND #Dept_Link_Internal.All_Selected_Running AND NOT #Dept_Link_Internal.All_Group_OFF THEN
       #StatusToECS := 2;
   END_IF;
   IF #AOn AND #Dept_Link_Internal.All_Group_OFF THEN #StatusToECS := 1; END_IF;
   IF #AOn AND #Dept_Link_Internal.All_Group_OFF AND #Dept_Link_Internal.All_Selected THEN
       #StatusToECS := 7;
   END_IF;
   IF #AOn AND #Dept_Link_Internal.MasterStop AND NOT #Dept_Link_Internal.All_Group_OFF THEN
       #StatusToECS := 4;
   END_IF;
   IF #AOn AND #Dept_Link_Internal.WatchDog_Failure AND NOT #Dept_Link_Internal.All_Group_OFF THEN
       #StatusToECS := 5;
   END_IF;
   IF #AOn AND #Dept_Link_Internal.QuickStop THEN #StatusToECS := 6; END_IF;
   IF #AOn AND NOT #STOP THEN #StatusToECS := 8; END_IF;
   IF #AOn AND NOT #DEMER THEN #StatusToECS := 200; END_IF;
END_REGION

REGION Network 20: Add Status to ECS status word
   // Bit 13 = 8192
   // Bit 12 = 4096
   // Bit 11 = 2048
   // Bit 10 = 1024
   // Bit  9 =  512
   // Bit  8 =  256
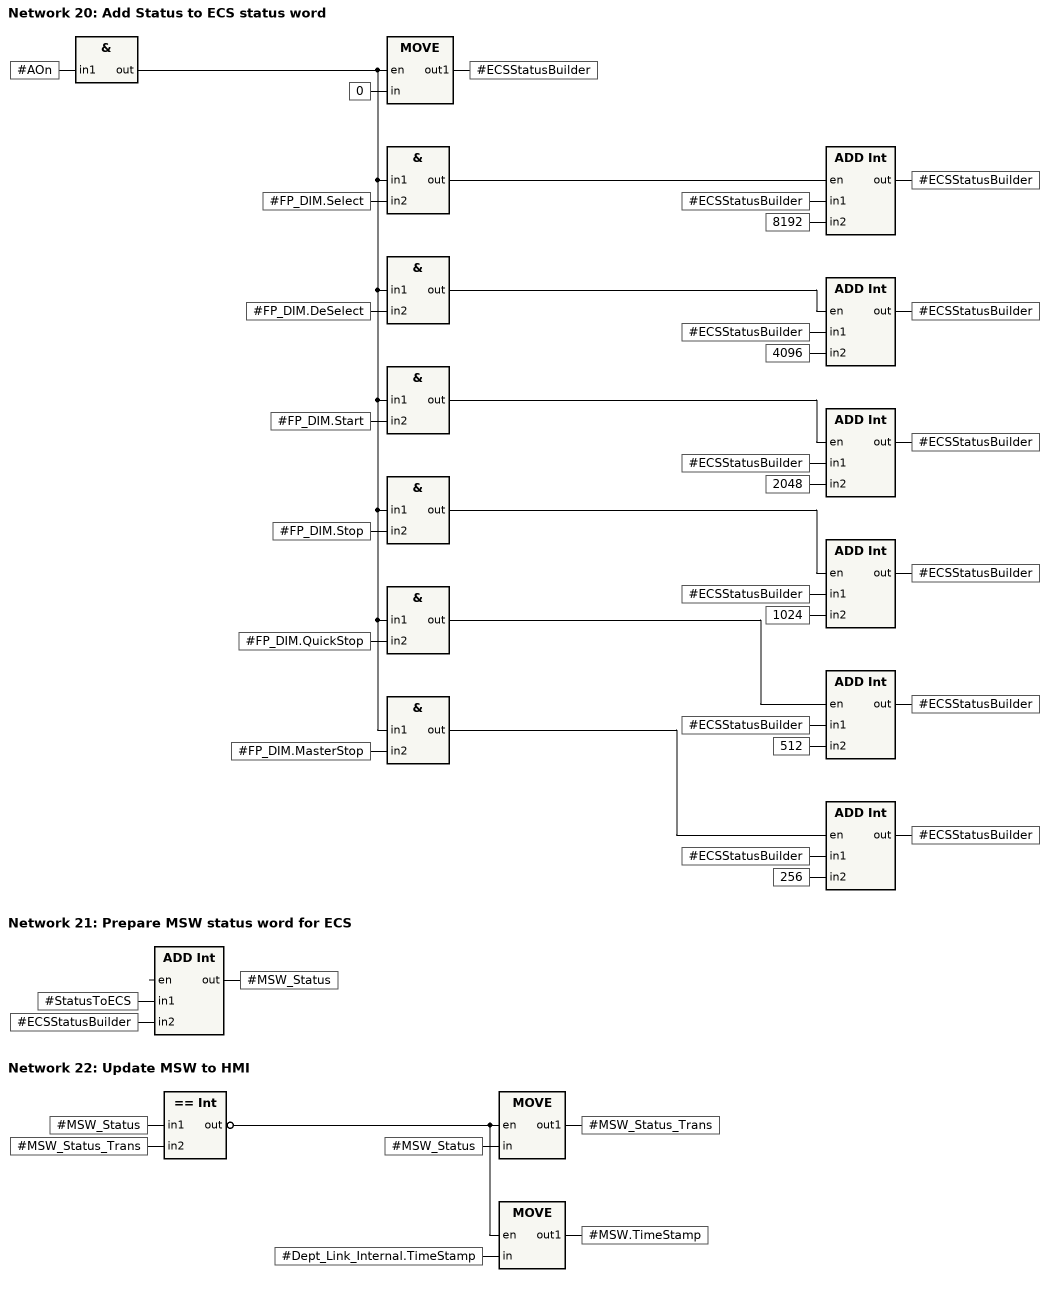
   IF #AOn THEN #ECSStatusBuilder := 0; END_IF;
   IF #AOn AND #FP_DIM.Select THEN #ECSStatusBuilder := #ECSStatusBuilder + 8192; END_IF;
   IF #AOn AND #FP_DIM.DeSelect THEN #ECSStatusBuilder := #ECSStatusBuilder + 4096; END_IF;
   IF #AOn AND #FP_DIM.Start THEN #ECSStatusBuilder := #ECSStatusBuilder + 2048; END_IF;
   IF #AOn AND #FP_DIM.Stop THEN #ECSStatusBuilder := #ECSStatusBuilder + 1024; END_IF;
   IF #AOn AND #FP_DIM.QuickStop THEN #ECSStatusBuilder := #ECSStatusBuilder + 512; END_IF;
   IF #AOn AND #FP_DIM.MasterStop THEN #ECSStatusBuilder := #ECSStatusBuilder + 256; END_IF;
END_REGION

REGION Network 21: Prepare MSW status word for ECS
   #MSW_Status := #StatusToECS + #ECSStatusBuilder;
END_REGION

REGION Network 22: Update MSW to HMI
   #_w1 := NOT (#MSW_Status = #MSW_Status_Trans);
   IF #_w1 THEN
       #MSW_Status_Trans := #MSW_Status;
       #MSW.TimeStamp := #Dept_Link_Internal.TimeStamp;
   END_IF;
END_REGION

REGION Network 23: Transfer MSW Internal to Actual Status Word
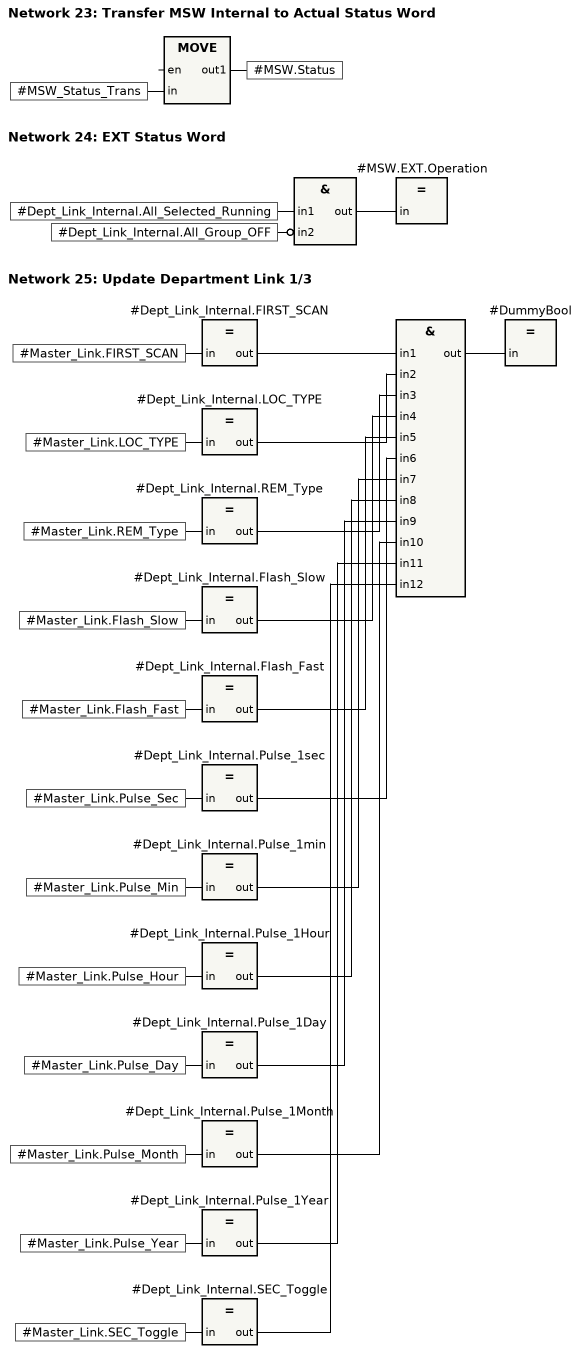
   #MSW.Status := #MSW_Status_Trans;
END_REGION

REGION Network 24: EXT Status Word
   #MSW.EXT.Operation := #Dept_Link_Internal.All_Selected_Running AND NOT #Dept_Link_Internal.All_Group_OFF;
END_REGION

REGION Network 25: Update Department Link 1/3
   #Dept_Link_Internal.FIRST_SCAN := #Master_Link.FIRST_SCAN;
   #Dept_Link_Internal.LOC_TYPE := #Master_Link.LOC_TYPE;
   #Dept_Link_Internal.REM_Type := #Master_Link.REM_Type;
   #Dept_Link_Internal.Flash_Slow := #Master_Link.Flash_Slow;
   #Dept_Link_Internal.Flash_Fast := #Master_Link.Flash_Fast;
   #Dept_Link_Internal.Pulse_1sec := #Master_Link.Pulse_Sec;
   #Dept_Link_Internal.Pulse_1min := #Master_Link.Pulse_Min;
   #Dept_Link_Internal.Pulse_1Hour := #Master_Link.Pulse_Hour;
   #Dept_Link_Internal.Pulse_1Day := #Master_Link.Pulse_Day;
   #Dept_Link_Internal.Pulse_1Month := #Master_Link.Pulse_Month;
   #Dept_Link_Internal.Pulse_1Year := #Master_Link.Pulse_Year;
   #Dept_Link_Internal.SEC_Toggle := #Master_Link.SEC_Toggle;
   #DummyBool := #Master_Link.FIRST_SCAN AND #Master_Link.LOC_TYPE AND #Master_Link.REM_Type AND #Master_Link.Flash_Slow AND #Master_Link.Flash_Fast AND #Master_Link.Pulse_Sec AND #Master_Link.Pulse_Min AND #Master_Link.Pulse_Hour AND #Master_Link.Pulse_Day AND #Master_Link.Pulse_Month AND #Master_Link.Pulse_Year AND #Master_Link.SEC_Toggle;
END_REGION

REGION Network 26: Update Department Link 2/3
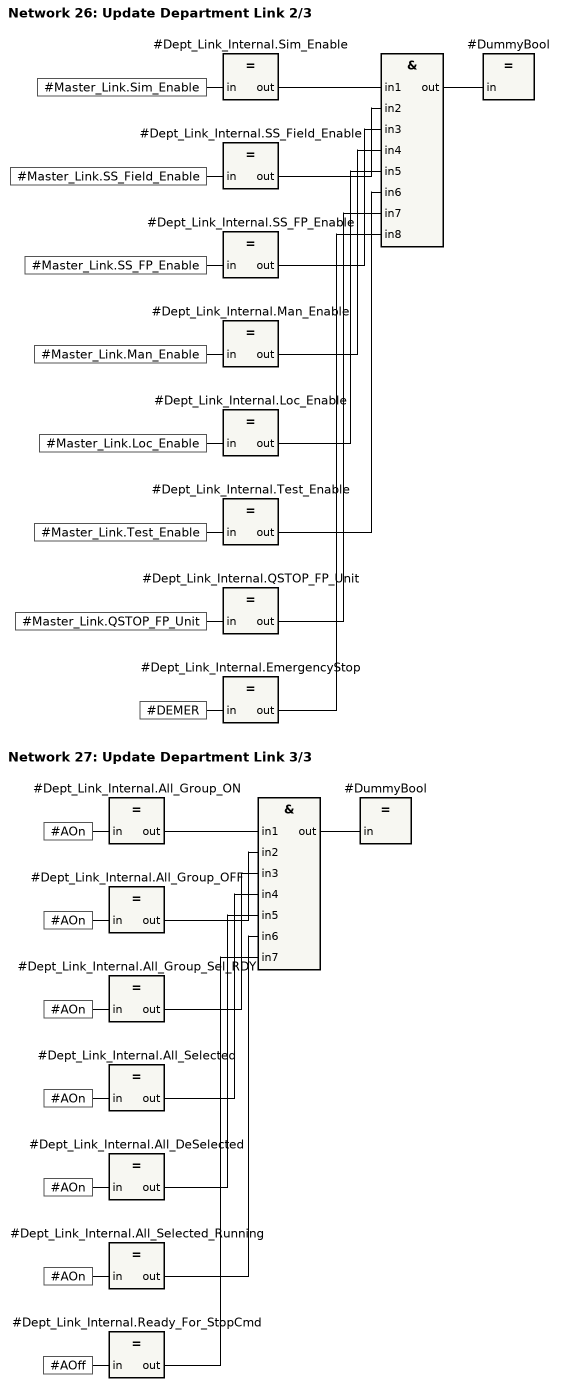
   #Dept_Link_Internal.Sim_Enable := #Master_Link.Sim_Enable;
   #Dept_Link_Internal.SS_Field_Enable := #Master_Link.SS_Field_Enable;
   #Dept_Link_Internal.SS_FP_Enable := #Master_Link.SS_FP_Enable;
   #Dept_Link_Internal.Man_Enable := #Master_Link.Man_Enable;
   #Dept_Link_Internal.Loc_Enable := #Master_Link.Loc_Enable;
   #Dept_Link_Internal.Test_Enable := #Master_Link.Test_Enable;
   #Dept_Link_Internal.QSTOP_FP_Unit := #Master_Link.QSTOP_FP_Unit;
   #Dept_Link_Internal.EmergencyStop := #DEMER;
   #DummyBool := #Master_Link.Sim_Enable AND #Master_Link.SS_Field_Enable AND #Master_Link.SS_FP_Enable AND #Master_Link.Man_Enable AND #Master_Link.Loc_Enable AND #Master_Link.Test_Enable AND #Master_Link.QSTOP_FP_Unit AND #DEMER;
END_REGION

REGION Network 27: Update Department Link 3/3
   #Dept_Link_Internal.All_Group_ON := #AOn;
   #Dept_Link_Internal.All_Group_OFF := #AOn;
   #Dept_Link_Internal.All_Group_Sel_RDY := #AOn;
   #Dept_Link_Internal.All_Selected := #AOn;
   #Dept_Link_Internal.All_DeSelected := #AOn;
   #Dept_Link_Internal.All_Selected_Running := #AOn;
   #Dept_Link_Internal.Ready_For_StopCmd := #AOff;
   #DummyBool := #AOn AND #AOn AND #AOn AND #AOn AND #AOn AND #AOn AND #AOff;
END_REGION

REGION Network 28: Transfer Depaetment Link Internal to Actual Dept Link
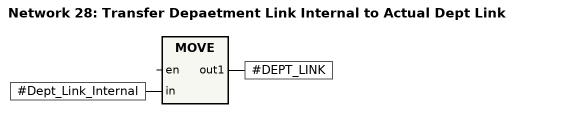
   #DEPT_LINK := #Dept_Link_Internal;
END_REGION
END_FUNCTION_BLOCK

FUNCTION_BLOCK "ACESYS_GROUP"   // FB202, FBD
TITLE = ACESYS V8.0 - Build 004 - GROUP Block
{ S7_Optimized_Access := 'FALSE' }
AUTHOR : FLSmidth
FAMILY : ACESYS
NAME : GROUP
VERSION : 8.0
   VAR_INPUT
      EnCtrl : Bool;   // Enable Control from Faceplate
      GRDY : Bool := TRUE;   // Group Ready
      GON : Bool := TRUE;   // Group On
      GOFF : Bool := TRUE;   // Group Off
      GSELD : Bool;   // Master Select
      GDSEL : Bool;   // Master De-select
      GEMER : Bool := TRUE;   // Group Emergency Stop
      START : Bool;   // Start from User Program
      STOP : Bool := TRUE;   // Stop from User Program
      RST : Bool;   // Reset from User Program
   END_VAR
   VAR_OUTPUT
      INTL : "ACESYS_INTL";   // Interlock
      INTL_SEQ_STR : "ACESYS_INTL";   // Interlock Sequence Start
      INTL_SEQ_STP : "ACESYS_INTL";   // Interlock Sequence Stop
      GSEL : Bool;   // Selected
      GSTR : Bool;   // Start
      GSTP : Bool;   // Stop
      GQSTP : Bool;   // Quick Stop
      GSS : Bool;   // Single Start
      GLTP : Bool;   // Local Test Permission
      GASTW : Bool;   // Start Warning Audioble
      GVSTW : Bool;   // Start Warning Visual
      GACC : Bool;   // Accepted
      GRUN : Bool;   // Running
      RESET : Bool;   // Reset Command
      RDY_START : Bool;   // Ready to Start
      GRP_OFF : Bool;   // Group is Off
      NOT_EMPTY : Bool;   // Not Empty, Material in Line
      CMD_OUT : "ACESYS_GRP_CMD";
      TOKEN : "ACESYS_TOKEN";
      MSW : "ACESYS_HMI_STAT_32T";
   END_VAR
   VAR_IN_OUT
      DEPT_LINK : "ACESYS_DEPT_LINK";
   END_VAR
   VAR
      BlockInfo : Struct
         Ace_Version : Int;   // Acesys Block Version Number
         Ace_BuildNo : Int;   // Acesys Block Build Number
         State_Act : Int;   // Actual State Number
         State_Prev : Int;   // Previous State Number
         DB_Number : Int;   // Block Instance DB Number
      END_STRUCT;
      FP_CMD : Struct   // Faceplate Commands
         Pause : Bool;
         RST_NotEmpty : Bool;
         Spare_11 : Bool;
         SS_Field : Bool;
         SelAndStart : Bool;
         DeselAndStop : Bool;
         Spare_14 : Bool;
         AckAlarm : Bool;
         Select : Bool;
         Auto : Bool;
         SS_FP : Bool;
         Local : Bool;
         Start : Bool;
         Stop : Bool;
         QuickStop : Bool;
         DeSelect : Bool;
      END_STRUCT;
      FP_SEL : Struct   // Faceplate Selections
         DeptCtrl : Bool;
         WD_LOCAL : Bool;
         Type_NoCtrl : Bool;
         NotEmpty : Bool;
         Spare12 : Bool;
         Spare11 : Bool;
         Spare10 : Bool;
         Spare09 : Bool;
         Spare08 : Bool;
         Spare07 : Bool;
         Spare06 : Bool;
         Spare05 : Bool;
         Spare04 : Bool;
         Spare03 : Bool;
         Spare02 : Bool;
         Spare01 : Bool;
      END_STRUCT;
      FP_DIM : Struct   // Faceplate Dimmed Buttons
         Select : Bool;
         Deselect : Bool;
         Start : Bool;
         Stop : Bool;
         QuickStop : Bool;
         Auto : Bool;
         Local : Bool;
         SS_FP : Bool;
         SS_Field : Bool;
         Pause : Bool;
         RST_NotEmpty : Bool;
         Spare5 : Bool;
         Spare4 : Bool;
         Spare3 : Bool;
         Spare2 : Bool;
         Spare1 : Bool;
      END_STRUCT;
      FP_SHOW : Struct   // Faceplate Show Buttons
         Auto : Bool;
         Local : Bool;
         SS_Field : Bool;
         SS_FP : Bool;
         NotEmpty : Bool;
         Spare11 : Bool;
         Spare10 : Bool;
         Spare09 : Bool;
         Spare08 : Bool;
         Spare07 : Bool;
         Spare06 : Bool;
         Spare05 : Bool;
         Spare04 : Bool;
         Spare03 : Bool;
         Spare02 : Bool;
         Spare01 : Bool;
      END_STRUCT;
      FP_PARM : Struct   // Faceplate Parameters
         StartWarn_Pre : Int;
         StartWarn_Acc : Int;
         StartFail_Pre : Int;
         StartFail_Acc : Int;
         StopFail_Pre : Int;
         StopFail_Acc : Int;
         StopReason : Int;
         SpareInt01 : Int;
         INTL : Bool;   // Interlock
         INTL_SEQ_STR : Bool;   // Interlock Sequence Start
         INTL_SEQ_STP : Bool;   // Interlock Sequence Stop
         Spare13 : Bool;
         Spare12 : Bool;
         Spare11 : Bool;
         Spare10 : Bool;
         Spare09 : Bool;
         Spare08 : Bool;
         Spare07 : Bool;
         Spare06 : Bool;
         Spare05 : Bool;
         Spare04 : Bool;
         Spare03 : Bool;
         Spare02 : Bool;
         Spare01 : Bool;
      END_STRUCT;
      STATE : Struct
         Stopped : Bool;
         WaitForSeqStop : Bool;
         QuickStop : Bool;
         Stopping : Bool;
         SingleStart_FP : Bool;
         SingleStart_Field : Bool;
         Selected : Bool;
         Accepted : Bool;
         WaitForSeqStart : Bool;
         StartWarning : Bool;
         Starting : Bool;
         Running : Bool;
         Pause : Bool;
         SelectedToStop : Bool;
         MasterStop : Bool;
         LocalMode : Bool;
         StopActive : Bool;
         EmergencyStop : Bool;
         NoCtrl : Bool;
         Alarm_Stop : Bool;
         Alarm_Start : Bool;
         NoStateActive : Bool;
         NoUnitSelected : Bool;
         Spare1 : Bool;
      END_STRUCT;
      ONS : Struct
         Cmd_Auto : Bool;
         Cmd_Local : Bool;
         Cmd_SS_FP : Bool;
         Cmd_SS_Field : Bool;
         START : Bool;
         RST : Bool;
         GSELD : Bool;
         GDSEL : Bool;
         Pause : Bool;
         SecPulse1 : Bool;
         SecPulse2 : Bool;
         Spare5 : Bool;
         Spare4 : Bool;
         Spare3 : Bool;
         Spare2 : Bool;
         Spare1 : Bool;
      END_STRUCT;
      StartWarn_Mem : Int;
      StartFail_Mem : Int;
      StopFail_Mem : Int;
      ModePointer : Int;
      AlarmNo : Int;
      AlarmNo_Old : Int;
      StatusWork : Int;
      ECSStatusBuilder : Int;
      MSW_Status : Int;
      ModeAuto : Bool;
      ModeLocal : Bool;
      ModeSS_Field : Bool;
      ModeSS_FP : Bool;
      StartWarn_Done : Bool;
      StartFail_Done : Bool;
      StopFail_Done : Bool;
      ALARM_AlarmPresent : Bool;
      ALARM_FailureAckRequired : Bool;
      CMD_Select : Bool;
      CMD_DeSelect : Bool;
      CMD_Start : Bool;
      CMD_Stop : Bool;
      CMD_QuickStop : Bool;
      CMD_AckAlarm : Bool;
      Sec_Pulse : Bool;
      RST_TMR : TOF_TIME;   // Delayed Reset CMD
      OUT : Struct
         GSEL : Bool;
         GSTR : Bool;
         GSTP : Bool;
         GQSTP : Bool;
         GSS : Bool;
         GLTP : Bool;
         GASTW : Bool;
         GVSTW : Bool;
         GACC : Bool;
         GRUN : Bool;
         RESET : Bool;
         RDY_START : Bool;
         GRP_OFF : Bool;
         NOT_EMPTY : Bool;
         INTL_OK_STAT : Bool;
         INTL_SEQ_STR_OK_STAT : Bool;
         INTL_SEQ_STP_OK_STAT : Bool;
      END_STRUCT;
      TOKEN_Stat : "ACESYS_TOKEN";
      MSW_Status_Trans : Int;
   END_VAR
   VAR_TEMP
      AOn : Bool;   // Always On
      AOff : Bool;   // Always Off
      DummyBool : Bool;
      CondForAccept : Bool;
      StatPointer_Old : Int;
      CMD_SelAndStart : Bool;
      CMD_DeselAndStop : Bool;
   END_VAR
   VAR_TEMP   // added for the SCL form of the ladder/FBD networks
      _w1 : Bool;
      _w2 : Bool;
      _w3 : Bool;
   END_VAR
BEGIN

REGION Network 1: Always On
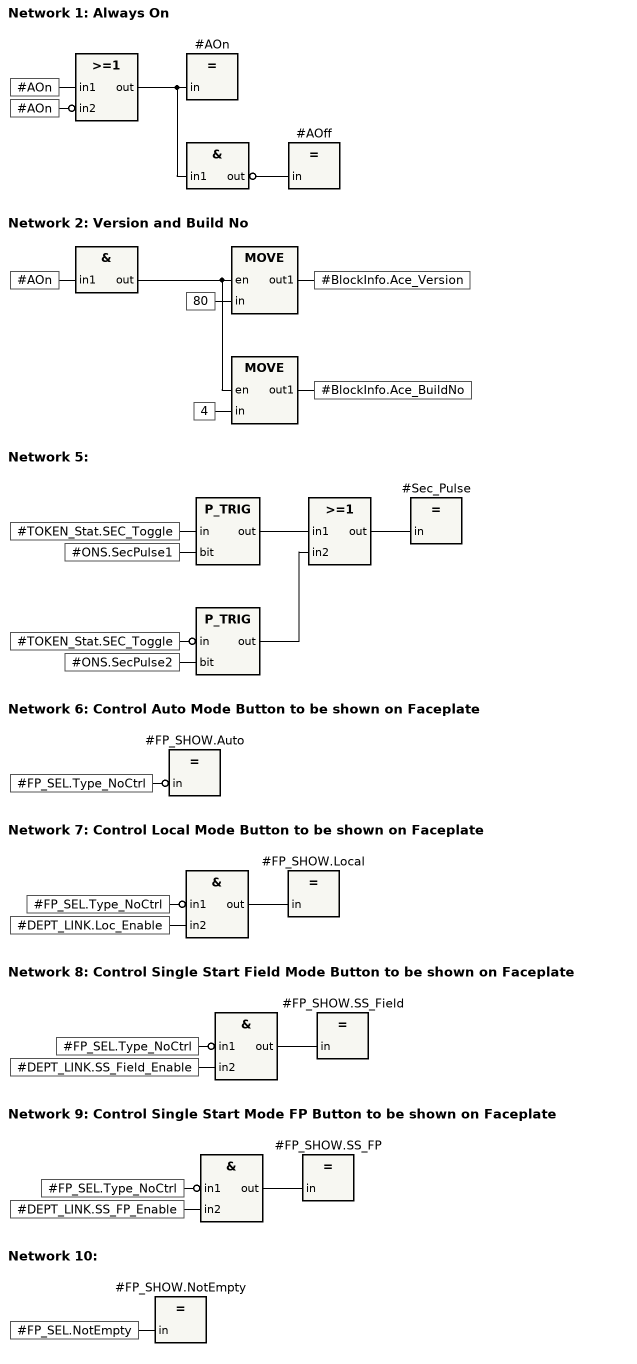
   #AOn := #AOn OR NOT #AOn;
   #AOff := NOT #AOn;
END_REGION

REGION Network 2: Version and Build No
   IF #AOn THEN
       #BlockInfo.Ace_Version := 80;
       #BlockInfo.Ace_BuildNo := 4;
   END_IF;
END_REGION

REGION Network 3 (STL): Instance DB Number to Faceplate
         L     DINO;
         T     #BlockInfo.DB_Number;
END_REGION

REGION Network 4 (SCL): Move Token to Token Stat
   #TOKEN_Stat.Acknowledge := PEEK_BOOL(area := 16#84, dbNumber := #BlockInfo.DB_Number, byteOffset := 16, bitOffset := 0);
   #TOKEN_Stat.AL_UNIT := PEEK_BOOL(area := 16#84, dbNumber := #BlockInfo.DB_Number, byteOffset := 16, bitOffset := 1);
   #TOKEN_Stat.StartWarn := PEEK_BOOL(area := 16#84, dbNumber := #BlockInfo.DB_Number, byteOffset := 16, bitOffset := 2);
   #TOKEN_Stat.GON := PEEK_BOOL(area := 16#84, dbNumber := #BlockInfo.DB_Number, byteOffset := 16, bitOffset := 3);
   #TOKEN_Stat.GOFF := PEEK_BOOL(area := 16#84, dbNumber := #BlockInfo.DB_Number, byteOffset := 16, bitOffset := 4);
   #TOKEN_Stat.Interlock_Unit := PEEK_BOOL(area := 16#84, dbNumber := #BlockInfo.DB_Number, byteOffset := 16, bitOffset := 5);
   #TOKEN_Stat.DeSelButRun := PEEK_BOOL(area := 16#84, dbNumber := #BlockInfo.DB_Number, byteOffset := 16, bitOffset := 6);
   #TOKEN_Stat.EmergencyStop := PEEK_BOOL(area := 16#84, dbNumber := #BlockInfo.DB_Number, byteOffset := 18, bitOffset := 0);
   #TOKEN_Stat.AllUnitsAuto := PEEK_BOOL(area := 16#84, dbNumber := #BlockInfo.DB_Number, byteOffset := 19, bitOffset := 2);
   #TOKEN_Stat.NotEmpty := PEEK_BOOL(area := 16#84, dbNumber := #BlockInfo.DB_Number, byteOffset := 19, bitOffset := 3);
   #TOKEN_Stat.SACK_On := PEEK_BOOL(area := 16#84, dbNumber := #BlockInfo.DB_Number, byteOffset := 19, bitOffset := 7);
   #TOKEN_Stat.SACK_Off := PEEK_BOOL(area := 16#84, dbNumber := #BlockInfo.DB_Number, byteOffset := 20, bitOffset := 0);
   #TOKEN_Stat.FIRST_SCAN := PEEK_BOOL(area := 16#84, dbNumber := #BlockInfo.DB_Number, byteOffset := 20, bitOffset := 1);
   #TOKEN_Stat.SEC_Toggle := PEEK_BOOL(area := 16#84, dbNumber := #BlockInfo.DB_Number, byteOffset := 20, bitOffset := 2);
   #TOKEN_Stat.UnitSelect := PEEK_BOOL(area := 16#84, dbNumber := #BlockInfo.DB_Number, byteOffset := 20, bitOffset := 3);
END_REGION

REGION Network 5
   #_w1 := #TOKEN_Stat.SEC_Toggle AND NOT #ONS.SecPulse1;   // rising edge
   #ONS.SecPulse1 := #TOKEN_Stat.SEC_Toggle;
   #_w2 := NOT #TOKEN_Stat.SEC_Toggle AND NOT #ONS.SecPulse2;   // rising edge
   #ONS.SecPulse2 := NOT #TOKEN_Stat.SEC_Toggle;
   #Sec_Pulse := #_w1 OR #_w2;
END_REGION

REGION Network 6: Control Auto Mode Button to be shown on Faceplate
   #FP_SHOW.Auto := NOT #FP_SEL.Type_NoCtrl;
END_REGION

REGION Network 7: Control Local Mode Button to be shown on Faceplate
   #FP_SHOW.Local := NOT #FP_SEL.Type_NoCtrl AND #DEPT_LINK.Loc_Enable;
END_REGION

REGION Network 8: Control Single Start Field Mode Button to be shown on Faceplate
   #FP_SHOW.SS_Field := NOT #FP_SEL.Type_NoCtrl AND #DEPT_LINK.SS_Field_Enable;
END_REGION

REGION Network 9: Control Single Start Mode FP Button to be shown on Faceplate
   #FP_SHOW.SS_FP := NOT #FP_SEL.Type_NoCtrl AND #DEPT_LINK.SS_FP_Enable;
END_REGION

REGION Network 10
   #FP_SHOW.NotEmpty := #FP_SEL.NotEmpty;
END_REGION

REGION Network 11: DIM SELECT Push Buttons on Faceplate
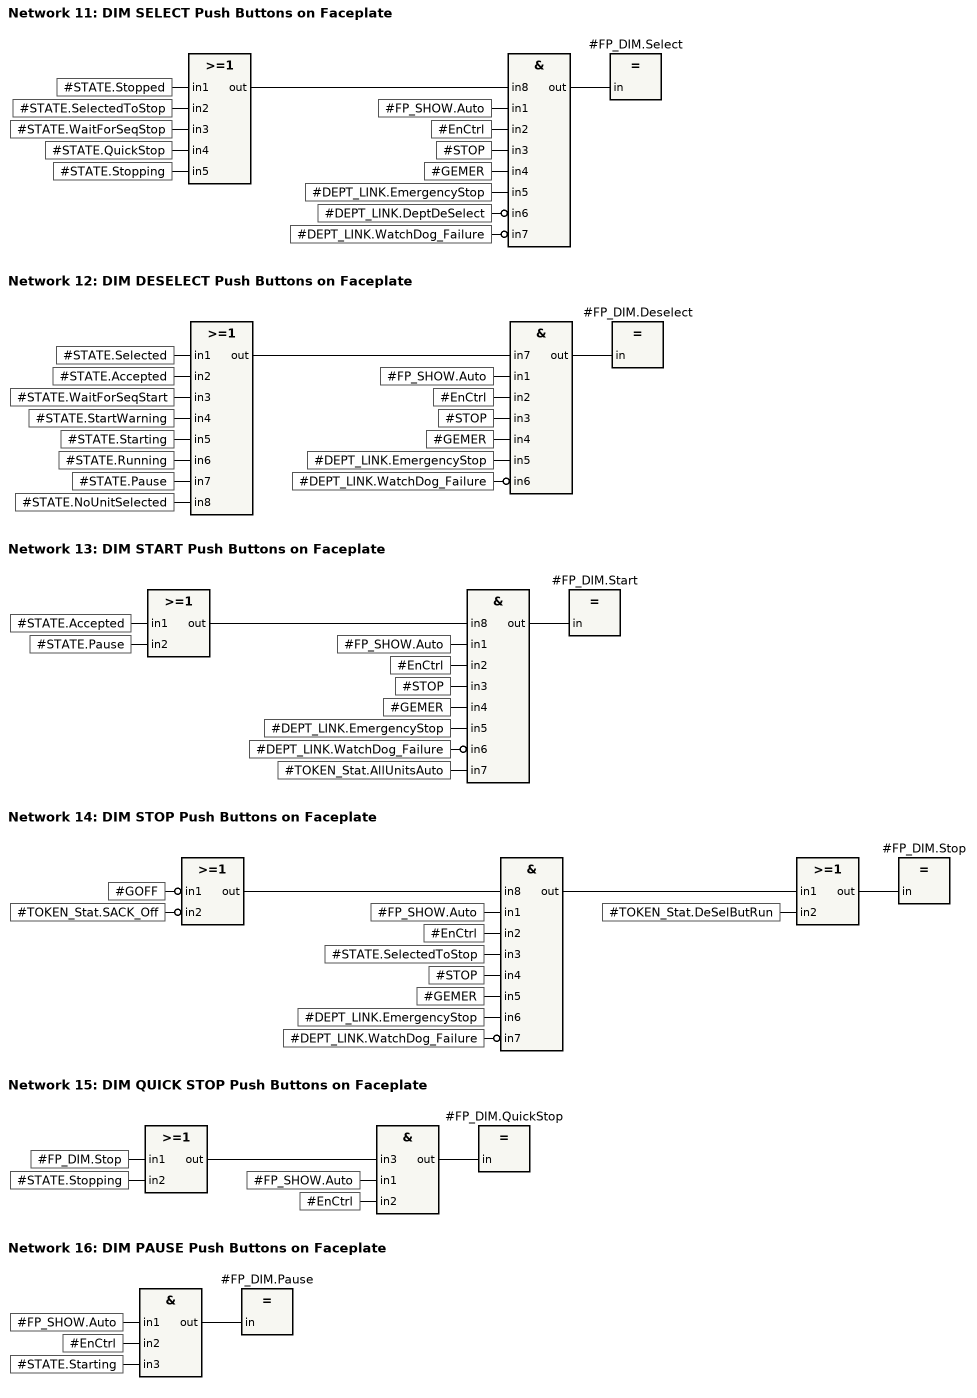
   #FP_DIM.Select := (#STATE.Stopped OR #STATE.SelectedToStop OR #STATE.WaitForSeqStop OR #STATE.QuickStop OR #STATE.Stopping) AND #FP_SHOW.Auto AND #EnCtrl AND #STOP AND #GEMER AND #DEPT_LINK.EmergencyStop AND NOT #DEPT_LINK.DeptDeSelect AND NOT #DEPT_LINK.WatchDog_Failure;
END_REGION

REGION Network 12: DIM DESELECT Push Buttons on Faceplate
   #FP_DIM.Deselect := (#STATE.Selected OR #STATE.Accepted OR #STATE.WaitForSeqStart OR #STATE.StartWarning OR #STATE.Starting OR #STATE.Running OR #STATE.Pause OR #STATE.NoUnitSelected) AND #FP_SHOW.Auto AND #EnCtrl AND #STOP AND #GEMER AND #DEPT_LINK.EmergencyStop AND NOT #DEPT_LINK.WatchDog_Failure;
END_REGION

REGION Network 13: DIM START Push Buttons on Faceplate
   #FP_DIM.Start := (#STATE.Accepted OR #STATE.Pause) AND #FP_SHOW.Auto AND #EnCtrl AND #STOP AND #GEMER AND #DEPT_LINK.EmergencyStop AND NOT #DEPT_LINK.WatchDog_Failure AND #TOKEN_Stat.AllUnitsAuto;
END_REGION

REGION Network 14: DIM STOP Push Buttons on Faceplate
   #FP_DIM.Stop := ((NOT #GOFF OR NOT #TOKEN_Stat.SACK_Off) AND #FP_SHOW.Auto AND #EnCtrl AND #STATE.SelectedToStop AND #STOP AND #GEMER AND #DEPT_LINK.EmergencyStop AND NOT #DEPT_LINK.WatchDog_Failure) OR #TOKEN_Stat.DeSelButRun;
END_REGION

REGION Network 15: DIM QUICK STOP Push Buttons on Faceplate
   #FP_DIM.QuickStop := (#FP_DIM.Stop OR #STATE.Stopping) AND #FP_SHOW.Auto AND #EnCtrl;
END_REGION

REGION Network 16: DIM PAUSE Push Buttons on Faceplate
   #FP_DIM.Pause := #FP_SHOW.Auto AND #EnCtrl AND #STATE.Starting;
END_REGION

REGION Network 17: DIM AUTO Push Buttons on Faceplate
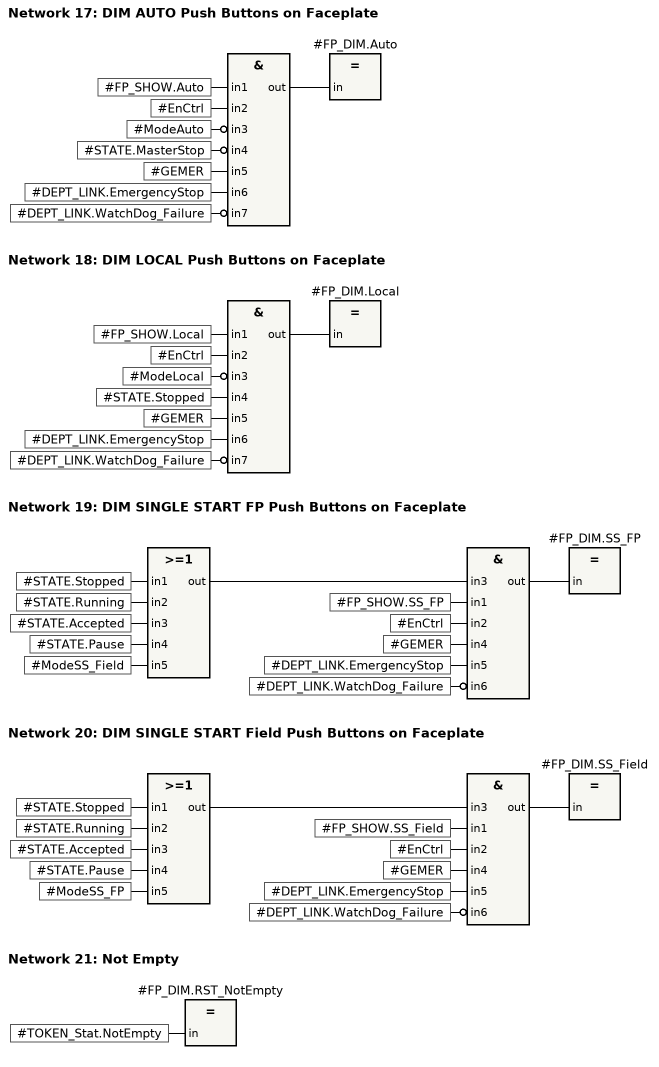
   #FP_DIM.Auto := #FP_SHOW.Auto AND #EnCtrl AND NOT #ModeAuto AND NOT #STATE.MasterStop AND #GEMER AND #DEPT_LINK.EmergencyStop AND NOT #DEPT_LINK.WatchDog_Failure;
END_REGION

REGION Network 18: DIM LOCAL Push Buttons on Faceplate
   #FP_DIM.Local := #FP_SHOW.Local AND #EnCtrl AND NOT #ModeLocal AND #STATE.Stopped AND #GEMER AND #DEPT_LINK.EmergencyStop AND NOT #DEPT_LINK.WatchDog_Failure;
END_REGION

REGION Network 19: DIM SINGLE START FP Push Buttons on Faceplate
   #FP_DIM.SS_FP := (#STATE.Stopped OR #STATE.Running OR #STATE.Accepted OR #STATE.Pause OR #ModeSS_Field) AND #FP_SHOW.SS_FP AND #EnCtrl AND #GEMER AND #DEPT_LINK.EmergencyStop AND NOT #DEPT_LINK.WatchDog_Failure;
END_REGION

REGION Network 20: DIM SINGLE START Field Push Buttons on Faceplate
   #FP_DIM.SS_Field := (#STATE.Stopped OR #STATE.Running OR #STATE.Accepted OR #STATE.Pause OR #ModeSS_FP) AND #FP_SHOW.SS_Field AND #EnCtrl AND #GEMER AND #DEPT_LINK.EmergencyStop AND NOT #DEPT_LINK.WatchDog_Failure;
END_REGION

REGION Network 21: Not Empty
   #FP_DIM.RST_NotEmpty := #TOKEN_Stat.NotEmpty;
END_REGION

REGION Network 22: Auto Mode
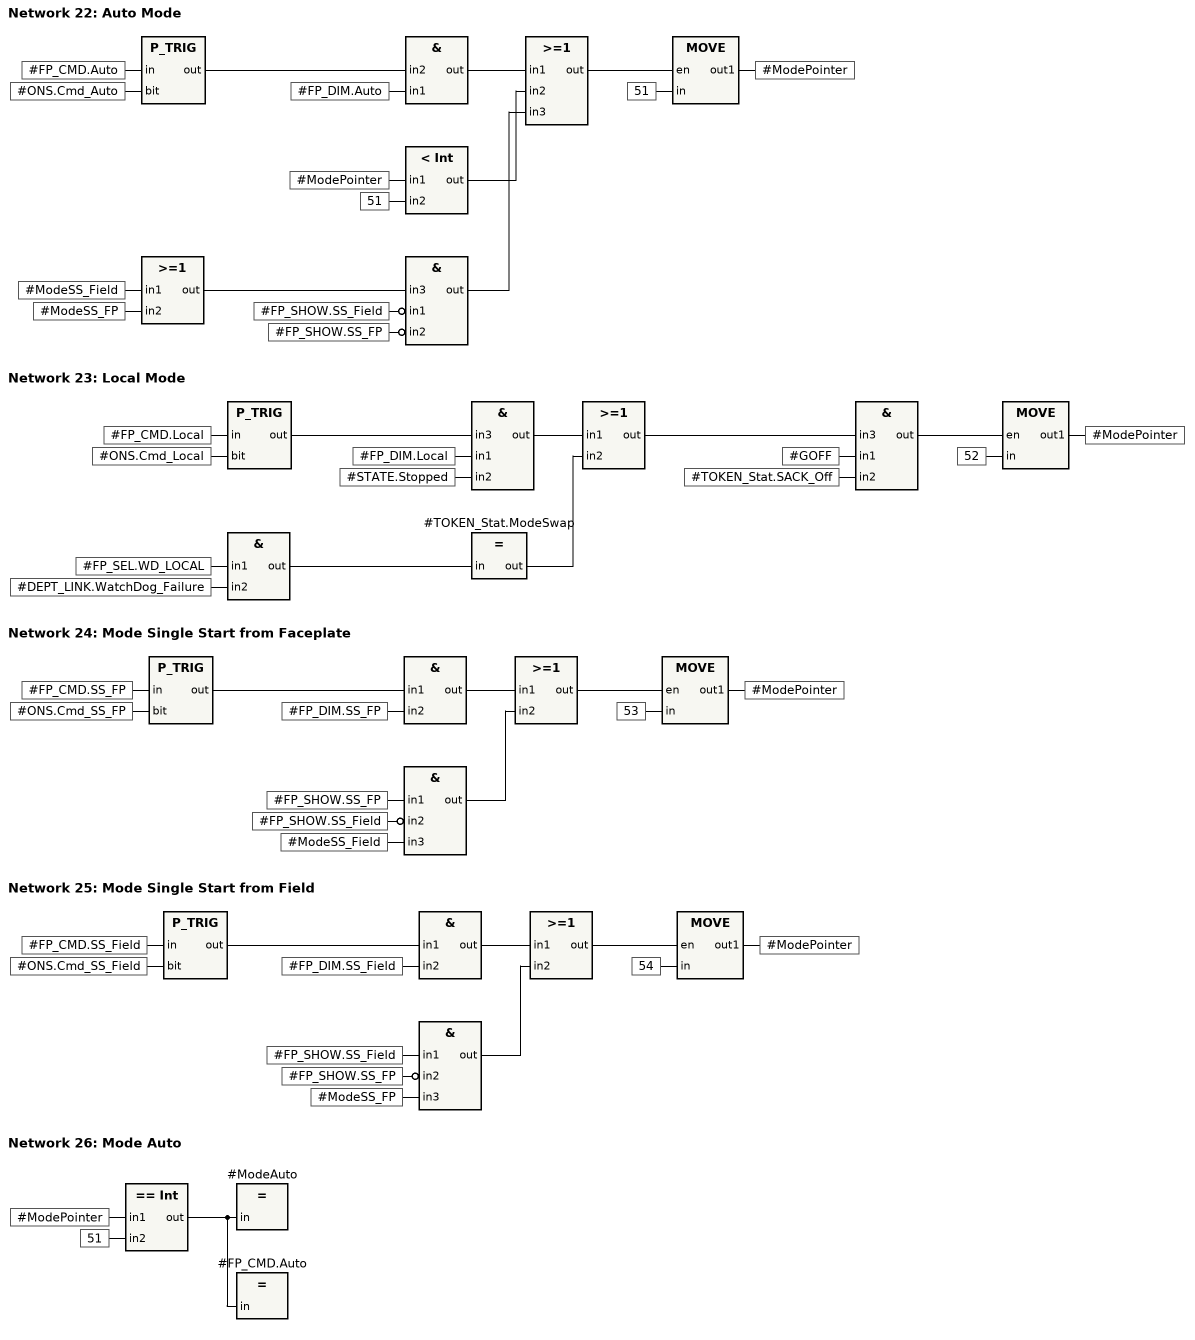
   #_w1 := #FP_CMD.Auto AND NOT #ONS.Cmd_Auto;   // rising edge
   #ONS.Cmd_Auto := #FP_CMD.Auto;
   IF (#_w1 AND #FP_DIM.Auto) OR (#ModePointer < 51) OR ((#ModeSS_Field OR #ModeSS_FP) AND NOT #FP_SHOW.SS_Field AND NOT #FP_SHOW.SS_FP) THEN
       #ModePointer := 51;
   END_IF;
END_REGION

REGION Network 23: Local Mode
   // Build 003 - 24.Jun.2020 (MIA-US): Removed TOKEN_Stat.SACK_On
   #_w1 := #FP_CMD.Local AND NOT #ONS.Cmd_Local;   // rising edge
   #ONS.Cmd_Local := #FP_CMD.Local;
   #TOKEN_Stat.ModeSwap := #FP_SEL.WD_LOCAL AND #DEPT_LINK.WatchDog_Failure;
   IF ((#_w1 AND #FP_DIM.Local AND #STATE.Stopped) OR #TOKEN_Stat.ModeSwap) AND #GOFF AND #TOKEN_Stat.SACK_Off THEN
       #ModePointer := 52;
   END_IF;
END_REGION

REGION Network 24: Mode Single Start from Faceplate
   #_w1 := #FP_CMD.SS_FP AND NOT #ONS.Cmd_SS_FP;   // rising edge
   #ONS.Cmd_SS_FP := #FP_CMD.SS_FP;
   IF (#_w1 AND #FP_DIM.SS_FP) OR (#FP_SHOW.SS_FP AND NOT #FP_SHOW.SS_Field AND #ModeSS_Field) THEN
       #ModePointer := 53;
   END_IF;
END_REGION

REGION Network 25: Mode Single Start from Field
   #_w1 := #FP_CMD.SS_Field AND NOT #ONS.Cmd_SS_Field;   // rising edge
   #ONS.Cmd_SS_Field := #FP_CMD.SS_Field;
   IF (#_w1 AND #FP_DIM.SS_Field) OR (#FP_SHOW.SS_Field AND NOT #FP_SHOW.SS_FP AND #ModeSS_FP) THEN
       #ModePointer := 54;
   END_IF;
END_REGION

REGION Network 26: Mode Auto
   #ModeAuto := #ModePointer = 51;
   #FP_CMD.Auto := #ModeAuto;
END_REGION

REGION Network 27: Mode Local
